KUKA KRL program: EPS_2_251825_SA29_A_20260116064109.src

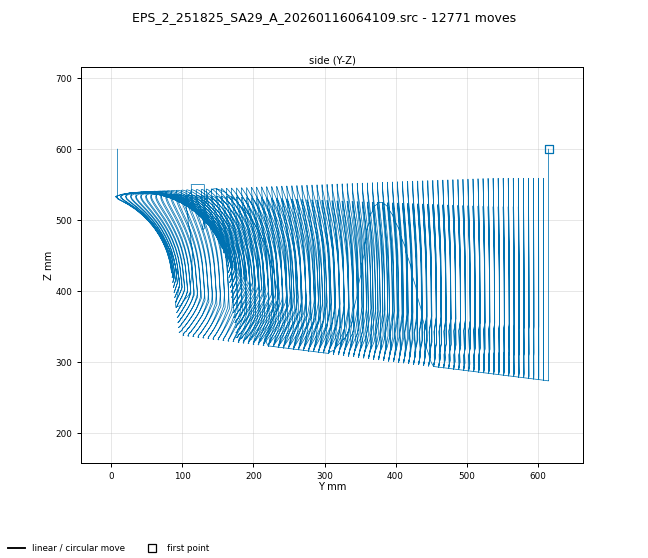
[picture p0: tool path of EPS_2_251825_SA29_A_20260116064109.src, 12771 of 12773 moves have a stored position in this frame; points joined in program order, loops and branches not executed]
&ACCESS RVP
&REL 4
&COMMENT QRS 19112012
&PARAM EDITMASK = *
DEF PART()
EXT BAS (BAS_COMMAND :IN,REAL :IN )
INT I
BAS (#INITMOV,0 )

;KUKA QRS Post kuka4.cps  Date:22-06-2017 !

File_ID=2988

QRS_PRE_INIT()

;Init var - Until changes are made in qrs_pre_init
Outlet_Square_prg=0
Inlet_1_Square_prg=0
Inlet_2_Square_prg=0
Inlet_3_Square_prg=0
Inlet_4_Square_prg=0
Inlet_5_Square_prg=0

Outlet_1={X 0.000, Y 535.490, Z 458.500, B 0.000, E1 0.000 }
Inlet_1={X 0.000, Y 538.340, Z 418.500, B 0.000, E1 195.000 }
Outlet_1_type=201
Inlet_1_type=201
;QRS#1=Sidecore dimensions
;QRS#2=200-8" PVC SDR 35
;QRS#3=200-8" PVC SDR 35
;QRS#4=
;QRS#5=
;QRS#6=
;QRS#7=
;QRS#8=
;QRS#9=12-08 PSX
;QRS#10=12-08 PSX
;QRS#11=
;QRS#12=
;QRS#13=
;QRS#14=
;QRS#15=
;QRS#16=1220x127x838 2,75'
;QRS#17=EPS Height
;QRS#18=559
;QRS#19=*
;QRS#20= UPDATED VERSION 22-06-2017
;QRS#21=*
Outlet_Square=0100
Inlet_1_Square=0100
Inlet_2_Square=0
Inlet_3_Square=0
Inlet_4_Square=0
Inlet_5_Square=0
Mill_Square=1
Outlet_Square_Prg=204
Inlet_1_Square_prg=204

QRS_INIT()

$ADVANCE=5

; T1
PTP {E1 173.613,E2 173.613}
PTP {X 0,Y 615.498,A -85,B 0,C 180,E1 173.613,E2 173.613,E3 0,E4 0,E5 0,E6 0}
QRS_SPEED_INIT()
LIN {X 0,Y 615.498,Z 600,A -85,B 0,C 180,E1 173.613,E2 173.613,E3 0,E4 0,E5 0,E6 0} C_VEL
LIN {X 0,Y 615.498,Z 283.876,A -85,B 0,C 180,E1 173.613,E2 173.613} C_VEL
LIN {X 0,Y 615.498,Z 275.694,A -85,B 0,C 180,E1 173.613,E2 173.613} C_VEL
LIN {X 0,Y 615.484,Z 273.694,A -85,B 0,C 180,E1 173.427,E2 173.427} C_VEL
LIN {X 0,Y 615.492,Z 273.68,A -85,B 0,C 180,E1 170.801,E2 170.801} C_VEL
LIN {X 0,Y 615.47,Z 273.687,A -85,B 0,C 180,E1 168.139,E2 168.139} C_VEL
LIN {X 0,Y 615.487,Z 273.702,A -85,B 0,C 180,E1 165.451,E2 165.451} C_VEL
LIN {X 0,Y 615.479,Z 273.686,A -85,B 0,C 180,E1 162.729,E2 162.729} C_VEL
LIN {X 0,Y 615.473,Z 273.685,A -85,B 0,C 180,E1 159.967,E2 159.967} C_VEL
LIN {X 0,Y 615.486,Z 273.703,A -85,B 0,C 180,E1 157.156,E2 157.156} C_VEL
LIN {X 0,Y 615.489,Z 273.681,A -85,B 0,C 180,E1 154.284,E2 154.284} C_VEL
LIN {X 0,Y 615.471,Z 273.688,A -85,B 0,C 180,E1 151.553,E2 151.553} C_VEL
LIN {X 0,Y 615.486,Z 273.702,A -85,B 0,C 180,E1 148.915,E2 148.915} C_VEL
LIN {X 0,Y 615.491,Z 273.68,A -85,B 0,C 180,E1 145.978,E2 145.978} C_VEL
LIN {X 0,Y 615.473,Z 273.692,A -85,B 0,C 180,E1 143.066,E2 143.066} C_VEL
LIN {X 0,Y 615.481,Z 273.692,A -85,B 0,C 180,E1 140.249,E2 140.249} C_VEL
LIN {X 0,Y 615.494,Z 273.679,A -85,B 0,C 180,E1 137.648,E2 137.648} C_VEL
LIN {X 0,Y 615.471,Z 273.689,A -85,B 0,C 180,E1 134.93,E2 134.93} C_VEL
LIN {X 0,Y 615.481,Z 273.695,A -85,B 0,C 180,E1 132.08,E2 132.08} C_VEL
LIN {X 0,Y 615.479,Z 273.688,A -85,B 0,C 180,E1 129.751,E2 129.751} C_VEL
LIN {X 0,Y 615.477,Z 273.684,A -85,B 0,C 180,E1 126.935,E2 126.935} C_VEL
LIN {X 0,Y 615.495,Z 273.7,A -85,B 0,C 180,E1 124.022,E2 124.022} C_VEL
LIN {X 0,Y 615.481,Z 273.682,A -85,B 0,C 180,E1 121.085,E2 121.085} C_VEL
LIN {X 0,Y 615.471,Z 273.688,A -85,B 0,C 180,E1 118.448,E2 118.448} C_VEL
LIN {X 0,Y 615.494,Z 273.699,A -85,B 0,C 180,E1 115.716,E2 115.716} C_VEL
LIN {X 0,Y 615.491,Z 273.68,A -85,B 0,C 180,E1 112.845,E2 112.845} C_VEL
LIN {X 0,Y 615.472,Z 273.691,A -85,B 0,C 180,E1 110.034,E2 110.034} C_VEL
LIN {X 0,Y 615.484,Z 273.694,A -85,B 0,C 180,E1 107.271,E2 107.271} C_VEL
LIN {X 0,Y 615.492,Z 273.68,A -85,B 0,C 180,E1 104.55,E2 104.55} C_VEL
LIN {X 0,Y 615.472,Z 273.689,A -85,B 0,C 180,E1 101.862,E2 101.862} C_VEL
LIN {X 0,Y 615.496,Z 273.699,A -85,B 0,C 180,E1 99.2,E2 99.2} C_VEL
LIN {X 0,Y 615.478,Z 273.686,A -85,B 0,C 180,E1 96.558,E2 96.558} C_VEL
LIN {X 0,Y 615.475,Z 273.685,A -85,B 0,C 180,E1 93.766,E2 93.766} C_VEL
LIN {X 0,Y 615.472,Z 273.814,A -85,B 0,C 180,E1 93.602,E2 93.602} C_VEL
LIN {X 0,Y 615.48,Z 289.251,A -85,B 0,C 180,E1 90.982,E2 90.982} C_VEL
LIN {X 0,Y 615.46,Z 304.876,A -85,B 0,C 180,E1 88.365,E2 88.365} C_VEL
LIN {X 0,Y 615.492,Z 308.179,A -85,B 0,C 180,E1 87.813,E2 87.813} C_VEL
LIN {X 0,Y 615.438,Z 414.942,A -85,B 0,C 180,E1 86.543,E2 86.543} C_VEL
LIN {X 0,Y 615.452,Z 427.227,A -85,B 0,C 180,E1 86.277,E2 86.277} C_VEL
LIN {X 0,Y 615.49,Z 439.928,A -85,B 0,C 180,E1 85.868,E2 85.868} C_VEL
LIN {X 0,Y 615.468,Z 452.119,A -85,B 0,C 180,E1 85.334,E2 85.334} C_VEL
LIN {X 0,Y 615.471,Z 463.598,A -85,B 0,C 180,E1 84.678,E2 84.678} C_VEL
LIN {X 0,Y 615.498,Z 473.921,A -85,B 0,C 180,E1 83.938,E2 83.938} C_VEL
LIN {X 0,Y 615.498,Z 481.714,A -85,B 0,C 180,E1 83.256,E2 83.256} C_VEL
LIN {X 0,Y 615.497,Z 489.534,A -85,B 0,C 180,E1 82.456,E2 82.456} C_VEL
LIN {X 0,Y 615.494,Z 497.406,A -85,B 0,C 180,E1 81.465,E2 81.465} C_VEL
LIN {X 0,Y 615.497,Z 503.699,A -85,B 0,C 180,E1 80.471,E2 80.471} C_VEL
LIN {X 0,Y 615.497,Z 508.721,A -85,B 0,C 180,E1 79.474,E2 79.474} C_VEL
LIN {X 0,Y 615.496,Z 512.609,A -85,B 0,C 180,E1 78.475,E2 78.475} C_VEL
LIN {X 0,Y 615.496,Z 515.466,A -85,B 0,C 180,E1 77.471,E2 77.471} C_VEL
LIN {X 0,Y 615.496,Z 516.804,A -85,B 0,C 180,E1 76.8,E2 76.8} C_VEL
LIN {X 0,Y 615.496,Z 517.816,A -85,B 0,C 180,E1 76.064,E2 76.064} C_VEL
LIN {X 0,Y 615.497,Z 518.274,A -85,B 0,C 180,E1 75.452,E2 75.452} C_VEL
LIN {X 0,Y 615.496,Z 518.351,A -85,B 0,C 180,E1 74.775,E2 74.775} C_VEL
LIN {X 0,Y 615.495,Z 517.486,A -85,B 0,C 180,E1 73.566,E2 73.566} C_VEL
LIN {X 0,Y 615.495,Z 516.099,A -85,B 0,C 180,E1 72.731,E2 72.731} C_VEL
LIN {X 0,Y 615.497,Z 514.451,A -85,B 0,C 180,E1 72.045,E2 72.045} C_VEL
LIN {X 0,Y 615.496,Z 511.079,A -85,B 0,C 180,E1 71.01,E2 71.01} C_VEL
LIN {X 0,Y 615.495,Z 506.514,A -85,B 0,C 180,E1 69.969,E2 69.969} C_VEL
LIN {X 0,Y 615.495,Z 500.595,A -85,B 0,C 180,E1 68.921,E2 68.921} C_VEL
LIN {X 0,Y 615.497,Z 492.996,A -85,B 0,C 180,E1 67.865,E2 67.865} C_VEL
LIN {X 0,Y 615.498,Z 485.049,A -85,B 0,C 180,E1 66.98,E2 66.98} C_VEL
LIN {X 0,Y 615.498,Z 476.915,A -85,B 0,C 180,E1 66.218,E2 66.218} C_VEL
LIN {X 0,Y 615.495,Z 467.048,A -85,B 0,C 180,E1 65.46,E2 65.46} C_VEL
LIN {X 0,Y 615.48,Z 456.212,A -85,B 0,C 180,E1 64.793,E2 64.793} C_VEL
LIN {X 0,Y 615.489,Z 443.762,A -85,B 0,C 180,E1 64.195,E2 64.195} C_VEL
LIN {X 0,Y 615.47,Z 431.051,A -85,B 0,C 180,E1 63.739,E2 63.739} C_VEL
LIN {X 0,Y 615.474,Z 418.085,A -85,B 0,C 180,E1 63.425,E2 63.425} C_VEL
LIN {X 0,Y 615.489,Z 400.248,A -85,B 0,C 180,E1 63.181,E2 63.181} C_VEL
LIN {X 0,Y 615.471,Z 308.115,A -85,B 0,C 180,E1 62.086,E2 62.086} C_VEL
LIN {X 0,Y 615.45,Z 292.43,A -85,B 0,C 180,E1 59.46,E2 59.46} C_VEL
LIN {X 0,Y 615.467,Z 276.486,A -85,B 0,C 180,E1 56.764,E2 56.764} C_VEL
LIN {X 0,Y 615.421,Z 273.7,A -85,B 0,C 180,E1 56.286,E2 56.286} C_VEL
LIN {X 0,Y 615.406,Z 273.7,A -85,B 0,C 180,E1 53.571,E2 53.571} C_VEL
LIN {X 0,Y 615.464,Z 273.7,A -85,B 0,C 180,E1 50.941,E2 50.941} C_VEL
LIN {X 0,Y 615.484,Z 273.698,A -85,B 0,C 180,E1 48.528,E2 48.528} C_VEL
LIN {X 0,Y 615.417,Z 273.698,A -85,B 0,C 180,E1 45.846,E2 45.846} C_VEL
LIN {X 0,Y 615.417,Z 273.699,A -85,B 0,C 180,E1 43.251,E2 43.251} C_VEL
LIN {X 0,Y 615.479,Z 273.7,A -85,B 0,C 180,E1 40.607,E2 40.607} C_VEL
LIN {X 0,Y 615.46,Z 273.695,A -85,B 0,C 180,E1 38.011,E2 38.011} C_VEL
LIN {X 0,Y 615.43,Z 273.695,A -85,B 0,C 180,E1 35.62,E2 35.62} C_VEL
LIN {X 0,Y 615.419,Z 273.696,A -85,B 0,C 180,E1 33.24,E2 33.24} C_VEL
LIN {X 0,Y 615.426,Z 273.697,A -85,B 0,C 180,E1 30.923,E2 30.923} C_VEL
LIN {X 0,Y 615.462,Z 273.699,A -85,B 0,C 180,E1 28.449,E2 28.449} C_VEL
LIN {X 0,Y 615.46,Z 273.692,A -85,B 0,C 180,E1 25.567,E2 25.567} C_VEL
LIN {X 0,Y 615.467,Z 273.691,A -85,B 0,C 180,E1 23.557,E2 23.557} C_VEL
LIN {X 0,Y 615.461,Z 273.691,A -85,B 0,C 180,E1 21.433,E2 21.433} C_VEL
LIN {X 0,Y 615.459,Z 273.69,A -85,B 0,C 180,E1 19.339,E2 19.339} C_VEL
LIN {X 0,Y 615.456,Z 273.691,A -85,B 0,C 180,E1 17.271,E2 17.271} C_VEL
LIN {X 0,Y 615.463,Z 273.689,A -85,B 0,C 180,E1 15.227,E2 15.227} C_VEL
LIN {X 0,Y 615.468,Z 273.688,A -85,B 0,C 180,E1 13.202,E2 13.202} C_VEL
LIN {X 0,Y 615.437,Z 273.693,A -85,B 0,C 180,E1 10.528,E2 10.528} C_VEL
LIN {X 0,Y 615.475,Z 273.698,A -85,B 0,C 180,E1 7.876,E2 7.876} C_VEL
LIN {X 0,Y 615.493,Z 273.688,A -85,B 0,C 180,E1 5.241,E2 5.241} C_VEL
LIN {X 0,Y 615.452,Z 273.689,A -85,B 0,C 180,E1 2.618,E2 2.618} C_VEL
LIN {X 0,Y 615.456,Z 273.688,A -85,B 0,C 180,E1 0.654,E2 0.654} C_VEL
LIN {X 0,Y 615.468,Z 273.686,A -85,B 0,C 180,E1 -1.309,E2 -1.309} C_VEL
LIN {X 0,Y 615.479,Z 273.685,A -85,B 0,C 180,E1 -3.273,E2 -3.273} C_VEL
LIN {X 0,Y 615.449,Z 273.691,A -85,B 0,C 180,E1 -5.899,E2 -5.899} C_VEL
LIN {X 0,Y 615.48,Z 273.698,A -85,B 0,C 180,E1 -8.537,E2 -8.537} C_VEL
LIN {X 0,Y 615.492,Z 273.687,A -85,B 0,C 180,E1 -11.193,E2 -11.193} C_VEL
LIN {X 0,Y 615.459,Z 273.687,A -85,B 0,C 180,E1 -13.929,E2 -13.929} C_VEL
LIN {X 0,Y 615.469,Z 273.696,A -85,B 0,C 180,E1 -16.587,E2 -16.587} C_VEL
LIN {X 0,Y 615.489,Z 273.689,A -85,B 0,C 180,E1 -19.338,E2 -19.338} C_VEL
LIN {X 0,Y 615.464,Z 273.686,A -85,B 0,C 180,E1 -22.138,E2 -22.138} C_VEL
LIN {X 0,Y 615.463,Z 273.687,A -85,B 0,C 180,E1 -24.273,E2 -24.273} C_VEL
LIN {X 0,Y 615.489,Z 273.699,A -85,B 0,C 180,E1 -27.049,E2 -27.049} C_VEL
LIN {X 0,Y 615.489,Z 273.684,A -85,B 0,C 180,E1 -29.798,E2 -29.798} C_VEL
LIN {X 0,Y 615.47,Z 273.685,A -85,B 0,C 180,E1 -32.459,E2 -32.459} C_VEL
LIN {X 0,Y 615.467,Z 273.691,A -85,B 0,C 180,E1 -34.817,E2 -34.817} C_VEL
LIN {X 0,Y 615.482,Z 273.698,A -85,B 0,C 180,E1 -37.243,E2 -37.243} C_VEL
LIN {X 0,Y 615.483,Z 273.685,A -85,B 0,C 180,E1 -40.091,E2 -40.091} C_VEL
LIN {X 0,Y 615.495,Z 273.68,A -85,B 0,C 180,E1 -42.353,E2 -42.353} C_VEL
LIN {X 0,Y 615.472,Z 273.69,A -85,B 0,C 180,E1 -45.07,E2 -45.07} C_VEL
LIN {X 0,Y 615.482,Z 273.694,A -85,B 0,C 180,E1 -47.921,E2 -47.921} C_VEL
LIN {X 0,Y 615.477,Z 273.688,A -85,B 0,C 180,E1 -50.251,E2 -50.251} C_VEL
LIN {X 0,Y 615.479,Z 273.684,A -85,B 0,C 180,E1 -53.065,E2 -53.065} C_VEL
LIN {X 0,Y 615.488,Z 273.697,A -85,B 0,C 180,E1 -55.98,E2 -55.98} C_VEL
LIN {X 0,Y 615.48,Z 273.682,A -85,B 0,C 180,E1 -58.916,E2 -58.916} C_VEL
LIN {X 0,Y 615.479,Z 273.69,A -85,B 0,C 180,E1 -61.552,E2 -61.552} C_VEL
LIN {X 0,Y 615.48,Z 273.695,A -85,B 0,C 180,E1 -64.285,E2 -64.285} C_VEL
LIN {X 0,Y 615.489,Z 273.68,A -85,B 0,C 180,E1 -67.157,E2 -67.157} C_VEL
LIN {X 0,Y 615.487,Z 273.758,A -85,B 0,C 180,E1 -67.438,E2 -67.438} C_VEL
LIN {X 0,Y 615.455,Z 293.701,A -85,B 0,C 180,E1 -70.141,E2 -70.141} C_VEL
LIN {X 0,Y 615.472,Z 313.086,A -85,B 0,C 180,E1 -72.73,E2 -72.73} C_VEL
LIN {X 0,Y 615.493,Z 334.924,A -85,B 0,C 180,E1 -75.607,E2 -75.607} C_VEL
LIN {X 0,Y 615.471,Z 346.477,A -85,B 0,C 180,E1 -77.114,E2 -77.114} C_VEL
LIN {X 0,Y 615.457,Z 454.9,A -85,B 0,C 180,E1 -78.411,E2 -78.411} C_VEL
LIN {X 0,Y 615.456,Z 467.391,A -85,B 0,C 180,E1 -78.682,E2 -78.682} C_VEL
LIN {X 0,Y 615.483,Z 480.688,A -85,B 0,C 180,E1 -79.116,E2 -79.116} C_VEL
LIN {X 0,Y 615.492,Z 492.498,A -85,B 0,C 180,E1 -79.641,E2 -79.641} C_VEL
LIN {X 0,Y 615.483,Z 504.013,A -85,B 0,C 180,E1 -80.305,E2 -80.305} C_VEL
LIN {X 0,Y 615.499,Z 514.355,A -85,B 0,C 180,E1 -81.051,E2 -81.051} C_VEL
LIN {X 0,Y 615.497,Z 522.703,A -85,B 0,C 180,E1 -81.795,E2 -81.795} C_VEL
LIN {X 0,Y 615.498,Z 530.615,A -85,B 0,C 180,E1 -82.621,E2 -82.621} C_VEL
LIN {X 0,Y 615.491,Z 538.211,A -85,B 0,C 180,E1 -83.609,E2 -83.609} C_VEL
LIN {X 0,Y 615.498,Z 545.21,A -85,B 0,C 180,E1 -84.76,E2 -84.76} C_VEL
LIN {X 0,Y 615.493,Z 549.856,A -85,B 0,C 180,E1 -85.745,E2 -85.745} C_VEL
LIN {X 0,Y 615.494,Z 553.402,A -85,B 0,C 180,E1 -86.728,E2 -86.728} C_VEL
LIN {X 0,Y 615.497,Z 555.235,A -85,B 0,C 180,E1 -87.383,E2 -87.383} C_VEL
LIN {X 0,Y 615.497,Z 556.61,A -85,B 0,C 180,E1 -88.038,E2 -88.038} C_VEL
LIN {X 0,Y 615.496,Z 558.174,A -85,B 0,C 180,E1 -89.347,E2 -89.347} C_VEL
LIN {X 0,Y 615.494,Z 558.389,A -85,B 0,C 180,E1 -90.001,E2 -90.001} C_VEL
LIN {X 0,Y 615.495,Z 557.579,A -85,B 0,C 180,E1 -91.31,E2 -91.31} C_VEL
LIN {X 0,Y 615.497,Z 556.607,A -85,B 0,C 180,E1 -91.964,E2 -91.964} C_VEL
LIN {X 0,Y 615.497,Z 555.23,A -85,B 0,C 180,E1 -92.619,E2 -92.619} C_VEL
LIN {X 0,Y 615.496,Z 552.346,A -85,B 0,C 180,E1 -93.602,E2 -93.602} C_VEL
LIN {X 0,Y 615.498,Z 548.438,A -85,B 0,C 180,E1 -94.585,E2 -94.585} C_VEL
LIN {X 0,Y 615.499,Z 543.4,A -85,B 0,C 180,E1 -95.571,E2 -95.571} C_VEL
LIN {X 0,Y 615.49,Z 536.913,A -85,B 0,C 180,E1 -96.578,E2 -96.578} C_VEL
LIN {X 0,Y 615.497,Z 529.125,A -85,B 0,C 180,E1 -97.546,E2 -97.546} C_VEL
LIN {X 0,Y 615.498,Z 519.247,A -85,B 0,C 180,E1 -98.537,E2 -98.537} C_VEL
LIN {X 0,Y 615.495,Z 508.853,A -85,B 0,C 180,E1 -99.365,E2 -99.365} C_VEL
LIN {X 0,Y 615.482,Z 498.561,A -85,B 0,C 180,E1 -100.029,E2 -100.029} C_VEL
LIN {X 0,Y 615.495,Z 487.122,A -85,B 0,C 180,E1 -100.617,E2 -100.617} C_VEL
LIN {X 0,Y 615.466,Z 475.341,A -85,B 0,C 180,E1 -101.078,E2 -101.078} C_VEL
LIN {X 0,Y 615.455,Z 462.209,A -85,B 0,C 180,E1 -101.445,E2 -101.445} C_VEL
LIN {X 0,Y 615.461,Z 448.878,A -85,B 0,C 180,E1 -101.674,E2 -101.674} C_VEL
LIN {X 0,Y 615.471,Z 346.462,A -85,B 0,C 180,E1 -102.888,E2 -102.888} C_VEL
LIN {X 0,Y 615.455,Z 325.984,A -85,B 0,C 180,E1 -105.567,E2 -105.567} C_VEL
LIN {X 0,Y 615.481,Z 305.471,A -85,B 0,C 180,E1 -108.282,E2 -108.282} C_VEL
LIN {X 0,Y 615.468,Z 283.338,A -85,B 0,C 180,E1 -111.258,E2 -111.258} C_VEL
LIN {X 0,Y 615.489,Z 273.682,A -85,B 0,C 180,E1 -112.594,E2 -112.594} C_VEL
LIN {X 0,Y 615.485,Z 273.681,A -85,B 0,C 180,E1 -114.993,E2 -114.993} C_VEL
LIN {X 0,Y 615.483,Z 273.698,A -85,B 0,C 180,E1 -117.916,E2 -117.916} C_VEL
LIN {X 0,Y 615.486,Z 273.682,A -85,B 0,C 180,E1 -120.921,E2 -120.921} C_VEL
LIN {X 0,Y 615.47,Z 273.686,A -85,B 0,C 180,E1 -123.531,E2 -123.531} C_VEL
LIN {X 0,Y 615.487,Z 273.7,A -85,B 0,C 180,E1 -126.425,E2 -126.425} C_VEL
LIN {X 0,Y 615.482,Z 273.685,A -85,B 0,C 180,E1 -129.061,E2 -129.061} C_VEL
LIN {X 0,Y 615.491,Z 273.68,A -85,B 0,C 180,E1 -131.474,E2 -131.474} C_VEL
LIN {X 0,Y 615.47,Z 273.691,A -85,B 0,C 180,E1 -134.152,E2 -134.152} C_VEL
LIN {X 0,Y 615.484,Z 273.693,A -85,B 0,C 180,E1 -136.954,E2 -136.954} C_VEL
LIN {X 0,Y 615.484,Z 273.684,A -85,B 0,C 180,E1 -139.393,E2 -139.393} C_VEL
LIN {X 0,Y 615.478,Z 273.683,A -85,B 0,C 180,E1 -141.99,E2 -141.99} C_VEL
LIN {X 0,Y 615.469,Z 273.689,A -85,B 0,C 180,E1 -144.383,E2 -144.383} C_VEL
LIN {X 0,Y 615.478,Z 273.695,A -85,B 0,C 180,E1 -146.763,E2 -146.763} C_VEL
LIN {X 0,Y 615.49,Z 273.702,A -85,B 0,C 180,E1 -149.08,E2 -149.08} C_VEL
LIN {X 0,Y 615.484,Z 273.681,A -85,B 0,C 180,E1 -152.085,E2 -152.085} C_VEL
LIN {X 0,Y 615.476,Z 273.683,A -85,B 0,C 180,E1 -154.434,E2 -154.434} C_VEL
LIN {X 0,Y 615.482,Z 273.696,A -85,B 0,C 180,E1 -157.155,E2 -157.155} C_VEL
LIN {X 0,Y 615.481,Z 273.687,A -85,B 0,C 180,E1 -159.967,E2 -159.967} C_VEL
LIN {X 0,Y 615.473,Z 273.684,A -85,B 0,C 180,E1 -162.729,E2 -162.729} C_VEL
LIN {X 0,Y 615.484,Z 273.697,A -85,B 0,C 180,E1 -165.451,E2 -165.451} C_VEL
LIN {X 0,Y 615.48,Z 273.69,A -85,B 0,C 180,E1 -168.139,E2 -168.139} C_VEL
LIN {X 0,Y 615.489,Z 273.68,A -85,B 0,C 180,E1 -170.801,E2 -170.801} C_VEL
LIN {X 0,Y 615.471,Z 273.691,A -85,B 0,C 180,E1 -173.443,E2 -173.443} C_VEL
LIN {X 0,Y 615.488,Z 273.699,A -85,B 0,C 180,E1 -176.071,E2 -176.071} C_VEL
LIN {X 0,Y 615.483,Z 273.684,A -85,B 0,C 180,E1 -178.691,E2 -178.691} C_VEL
LIN {X 0,Y 615.478,Z 273.683,A -85,B 0,C 180,E1 -181.308,E2 -181.308} C_VEL
LIN {X 0,Y 615.476,Z 273.694,A -85,B 0,C 180,E1 -183.928,E2 -183.928} C_VEL
LIN {X 0,Y 615.484,Z 273.694,A -85,B 0,C 180,E1 -186.573,E2 -186.573} C_VEL
LIN {X 0,Y 614.811,Z 273.83,A -85,B 0,C 180,E1 -187.118,E2 -187.118} C_VEL
LIN {X 0,Y 611.983,Z 274.251,A -85,B 0,C 180,E1 -188.004,E2 -188.004} C_VEL
LIN {X 0,Y 609.592,Z 274.558,A -85,B 0,C 180,E1 -188.717,E2 -188.717} C_VEL
LIN {X 0,Y 608.552,Z 274.675,A -85,B 0,C 180,E1 -189.267,E2 -189.267} C_VEL
LIN {X 0,Y 608.459,Z 274.685,A -85,B 0,C 180,E1 -189.453,E2 -189.453} C_VEL
LIN {X 0,Y 608.452,Z 274.689,A -85,B 0,C 180,E1 -192,E2 -192} C_VEL
LIN {X 0,Y 608.475,Z 274.693,A -85,B 0,C 180,E1 -194.72,E2 -194.72} C_VEL
LIN {X 0,Y 608.446,Z 274.688,A -85,B 0,C 180,E1 -197.477,E2 -197.477} C_VEL
LIN {X 0,Y 608.446,Z 274.687,A -85,B 0,C 180,E1 -199.571,E2 -199.571} C_VEL
LIN {X 0,Y 608.46,Z 274.685,A -85,B 0,C 180,E1 -201.692,E2 -201.692} C_VEL
LIN {X 0,Y 608.448,Z 274.692,A -85,B 0,C 180,E1 -204.571,E2 -204.571} C_VEL
LIN {X 0,Y 608.482,Z 274.69,A -85,B 0,C 180,E1 -207.207,E2 -207.207} C_VEL
LIN {X 0,Y 608.468,Z 274.684,A -85,B 0,C 180,E1 -209.971,E2 -209.971} C_VEL
LIN {X 0,Y 608.453,Z 274.692,A -85,B 0,C 180,E1 -212.88,E2 -212.88} C_VEL
LIN {X 0,Y 608.436,Z 274.7,A -85,B 0,C 180,E1 -215.278,E2 -215.278} C_VEL
LIN {X 0,Y 608.468,Z 274.689,A -85,B 0,C 180,E1 -217.746,E2 -217.746} C_VEL
LIN {X 0,Y 608.446,Z 274.687,A -85,B 0,C 180,E1 -220.328,E2 -220.328} C_VEL
LIN {X 0,Y 608.441,Z 274.69,A -85,B 0,C 180,E1 -222.961,E2 -222.961} C_VEL
LIN {X 0,Y 608.453,Z 274.695,A -85,B 0,C 180,E1 -225.736,E2 -225.736} C_VEL
LIN {X 0,Y 608.462,Z 274.685,A -85,B 0,C 180,E1 -228.658,E2 -228.658} C_VEL
LIN {X 0,Y 608.469,Z 274.695,A -85,B 0,C 180,E1 -231.759,E2 -231.759} C_VEL
LIN {X 0,Y 608.447,Z 274.697,A -85,B 0,C 180,E1 -233.954,E2 -233.954} C_VEL
LIN {X 0,Y 608.45,Z 274.691,A -85,B 0,C 180,E1 -236.328,E2 -236.328} C_VEL
LIN {X 0,Y 608.448,Z 274.688,A -85,B 0,C 180,E1 -238.732,E2 -238.732} C_VEL
LIN {X 0,Y 608.464,Z 274.686,A -85,B 0,C 180,E1 -241.382,E2 -241.382} C_VEL
LIN {X 0,Y 608.444,Z 274.694,A -85,B 0,C 180,E1 -243.964,E2 -243.964} C_VEL
LIN {X 0,Y 608.454,Z 274.688,A -85,B 0,C 180,E1 -246.875,E2 -246.875} C_VEL
LIN {X 0,Y 608.455,Z 274.687,A -85,B 0,C 180,E1 -249.725,E2 -249.725} C_VEL
LIN {X 0,Y 608.442,Z 274.689,A -85,B 0,C 180,E1 -251.827,E2 -251.827} C_VEL
LIN {X 0,Y 608.466,Z 274.696,A -85,B 0,C 180,E1 -254.593,E2 -254.593} C_VEL
LIN {X 0,Y 608.475,Z 274.685,A -85,B 0,C 180,E1 -257.322,E2 -257.322} C_VEL
LIN {X 0,Y 608.445,Z 274.688,A -85,B 0,C 180,E1 -260.022,E2 -260.022} C_VEL
LIN {X 0,Y 608.464,Z 274.694,A -85,B 0,C 180,E1 -262.7,E2 -262.7} C_VEL
LIN {X 0,Y 608.448,Z 274.691,A -85,B 0,C 180,E1 -265.361,E2 -265.361} C_VEL
LIN {X 0,Y 608.459,Z 274.691,A -85,B 0,C 180,E1 -266.315,E2 -266.315} C_VEL
LIN {X 0,Y 608.494,Z 288.467,A -85,B 0,C 180,E1 -268.675,E2 -268.675} C_VEL
LIN {X 0,Y 608.44,Z 304.132,A -85,B 0,C 180,E1 -271.323,E2 -271.323} C_VEL
LIN {X 0,Y 608.493,Z 308.629,A -85,B 0,C 180,E1 -272.047,E2 -272.047} C_VEL
LIN {X 0,Y 608.484,Z 415.486,A -85,B 0,C 180,E1 -273.33,E2 -273.33} C_VEL
LIN {X 0,Y 608.496,Z 429.112,A -85,B 0,C 180,E1 -273.641,E2 -273.641} C_VEL
LIN {X 0,Y 608.528,Z 441.372,A -85,B 0,C 180,E1 -274.055,E2 -274.055} C_VEL
LIN {X 0,Y 608.474,Z 452.439,A -85,B 0,C 180,E1 -274.553,E2 -274.553} C_VEL
LIN {X 0,Y 608.457,Z 463.926,A -85,B 0,C 180,E1 -275.218,E2 -275.218} C_VEL
LIN {X 0,Y 608.498,Z 474.271,A -85,B 0,C 180,E1 -275.965,E2 -275.965} C_VEL
LIN {X 0,Y 608.478,Z 481.861,A -85,B 0,C 180,E1 -276.631,E2 -276.631} C_VEL
LIN {X 0,Y 608.47,Z 489.951,A -85,B 0,C 180,E1 -277.465,E2 -277.465} C_VEL
LIN {X 0,Y 608.44,Z 497.87,A -85,B 0,C 180,E1 -278.468,E2 -278.468} C_VEL
LIN {X 0,Y 608.437,Z 503.247,A -85,B 0,C 180,E1 -279.305,E2 -279.305} C_VEL
LIN {X 0,Y 608.459,Z 508.516,A -85,B 0,C 180,E1 -280.312,E2 -280.312} C_VEL
LIN {X 0,Y 608.427,Z 512.617,A -85,B 0,C 180,E1 -281.324,E2 -281.324} C_VEL
LIN {X 0,Y 608.439,Z 514.749,A -85,B 0,C 180,E1 -281.999,E2 -281.999} C_VEL
LIN {X 0,Y 608.419,Z 516.43,A -85,B 0,C 180,E1 -282.677,E2 -282.677} C_VEL
LIN {X 0,Y 608.438,Z 517.694,A -85,B 0,C 180,E1 -283.356,E2 -283.356} C_VEL
LIN {X 0,Y 608.421,Z 518.539,A -85,B 0,C 180,E1 -284.037,E2 -284.037} C_VEL
LIN {X 0,Y 608.418,Z 518.93,A -85,B 0,C 180,E1 -284.721,E2 -284.721} C_VEL
LIN {X 0,Y 608.418,Z 518.921,A -85,B 0,C 180,E1 -285.406,E2 -285.406} C_VEL
LIN {X 0,Y 608.423,Z 518.012,A -85,B 0,C 180,E1 -286.515,E2 -286.515} C_VEL
LIN {X 0,Y 608.42,Z 516.293,A -85,B 0,C 180,E1 -287.476,E2 -287.476} C_VEL
LIN {X 0,Y 608.428,Z 512.84,A -85,B 0,C 180,E1 -288.704,E2 -288.704} C_VEL
LIN {X 0,Y 608.434,Z 507.819,A -85,B 0,C 180,E1 -289.921,E2 -289.921} C_VEL
LIN {X 0,Y 608.45,Z 502.058,A -85,B 0,C 180,E1 -290.98,E2 -290.98} C_VEL
LIN {X 0,Y 608.454,Z 494.729,A -85,B 0,C 180,E1 -292.047,E2 -292.047} C_VEL
LIN {X 0,Y 608.456,Z 487.093,A -85,B 0,C 180,E1 -292.942,E2 -292.942} C_VEL
LIN {X 0,Y 608.481,Z 477.658,A -85,B 0,C 180,E1 -293.843,E2 -293.843} C_VEL
LIN {X 0,Y 608.493,Z 467.137,A -85,B 0,C 180,E1 -294.659,E2 -294.659} C_VEL
LIN {X 0,Y 608.48,Z 455.524,A -85,B 0,C 180,E1 -295.371,E2 -295.371} C_VEL
LIN {X 0,Y 608.517,Z 443.797,A -85,B 0,C 180,E1 -295.934,E2 -295.934} C_VEL
LIN {X 0,Y 608.515,Z 432.326,A -85,B 0,C 180,E1 -296.353,E2 -296.353} C_VEL
LIN {X 0,Y 608.539,Z 419.33,A -85,B 0,C 180,E1 -296.687,E2 -296.687} C_VEL
LIN {X 0,Y 608.539,Z 403.321,A -85,B 0,C 180,E1 -296.921,E2 -296.921} C_VEL
LIN {X 0,Y 608.431,Z 308.378,A -85,B 0,C 180,E1 -298.055,E2 -298.055} C_VEL
LIN {X 0,Y 608.451,Z 293.599,A -85,B 0,C 180,E1 -300.544,E2 -300.544} C_VEL
LIN {X 0,Y 608.454,Z 276.455,A -85,B 0,C 180,E1 -303.471,E2 -303.471} C_VEL
LIN {X 0,Y 608.403,Z 274.695,A -85,B 0,C 180,E1 -303.79,E2 -303.79} C_VEL
LIN {X 0,Y 608.375,Z 274.696,A -85,B 0,C 180,E1 -306.095,E2 -306.095} C_VEL
LIN {X 0,Y 608.375,Z 274.696,A -85,B 0,C 180,E1 -308.229,E2 -308.229} C_VEL
LIN {X 0,Y 608.39,Z 274.694,A -85,B 0,C 180,E1 -310.322,E2 -310.322} C_VEL
LIN {X 0,Y 608.379,Z 274.696,A -85,B 0,C 180,E1 -312.326,E2 -312.326} C_VEL
LIN {X 0,Y 608.394,Z 274.694,A -85,B 0,C 180,E1 -314.258,E2 -314.258} C_VEL
LIN {X 0,Y 608.412,Z 274.692,A -85,B 0,C 180,E1 -316.695,E2 -316.695} C_VEL
LIN {X 0,Y 608.391,Z 274.695,A -85,B 0,C 180,E1 -318.818,E2 -318.818} C_VEL
LIN {X 0,Y 608.405,Z 274.701,A -85,B 0,C 180,E1 -321.407,E2 -321.407} C_VEL
LIN {X 0,Y 608.428,Z 274.695,A -85,B 0,C 180,E1 -323.954,E2 -323.954} C_VEL
LIN {X 0,Y 608.428,Z 274.691,A -85,B 0,C 180,E1 -326.327,E2 -326.327} C_VEL
LIN {X 0,Y 608.415,Z 274.691,A -85,B 0,C 180,E1 -328.734,E2 -328.734} C_VEL
LIN {X 0,Y 608.441,Z 274.692,A -85,B 0,C 180,E1 -331.382,E2 -331.382} C_VEL
LIN {X 0,Y 608.456,Z 274.69,A -85,B 0,C 180,E1 -334.278,E2 -334.278} C_VEL
LIN {X 0,Y 608.412,Z 274.692,A -85,B 0,C 180,E1 -336.875,E2 -336.875} C_VEL
LIN {X 0,Y 608.425,Z 274.691,A -85,B 0,C 180,E1 -339.327,E2 -339.327} C_VEL
LIN {X 0,Y 608.436,Z 274.696,A -85,B 0,C 180,E1 -341.828,E2 -341.828} C_VEL
LIN {X 0,Y 608.454,Z 274.69,A -85,B 0,C 180,E1 -344.594,E2 -344.594} C_VEL
LIN {X 0,Y 608.435,Z 274.689,A -85,B 0,C 180,E1 -347.322,E2 -347.322} C_VEL
LIN {X 0,Y 608.444,Z 274.694,A -85,B 0,C 180,E1 -350.023,E2 -350.023} C_VEL
LIN {X 0,Y 608.475,Z 274.688,A -85,B 0,C 180,E1 -352.701,E2 -352.701} C_VEL
LIN {X 0,Y 608.418,Z 274.691,A -85,B 0,C 180,E1 -355.362,E2 -355.362} C_VEL
LIN {X 0,Y 608.446,Z 274.687,A -85,B 0,C 180,E1 -357.352,E2 -357.352} C_VEL
LIN {X 0,Y 608.443,Z 274.691,A -85,B 0,C 180,E1 -360,E2 -360} C_VEL
LIN {X 0,Y 608.485,Z 274.692,A -85,B 0,C 180,E1 -362.648,E2 -362.648} C_VEL
LIN {X 0,Y 608.461,Z 274.687,A -85,B 0,C 180,E1 -365.302,E2 -365.302} C_VEL
LIN {X 0,Y 608.449,Z 274.688,A -85,B 0,C 180,E1 -367.967,E2 -367.967} C_VEL
LIN {X 0,Y 608.458,Z 274.695,A -85,B 0,C 180,E1 -370.65,E2 -370.65} C_VEL
LIN {X 0,Y 608.461,Z 274.688,A -85,B 0,C 180,E1 -373.357,E2 -373.357} C_VEL
LIN {X 0,Y 608.438,Z 274.689,A -85,B 0,C 180,E1 -376.095,E2 -376.095} C_VEL
LIN {X 0,Y 608.445,Z 274.698,A -85,B 0,C 180,E1 -378.87,E2 -378.87} C_VEL
LIN {X 0,Y 608.459,Z 274.687,A -85,B 0,C 180,E1 -381.692,E2 -381.692} C_VEL
LIN {X 0,Y 608.441,Z 274.691,A -85,B 0,C 180,E1 -384.572,E2 -384.572} C_VEL
LIN {X 0,Y 608.478,Z 274.694,A -85,B 0,C 180,E1 -387.211,E2 -387.211} C_VEL
LIN {X 0,Y 608.467,Z 274.685,A -85,B 0,C 180,E1 -389.975,E2 -389.975} C_VEL
LIN {X 0,Y 608.446,Z 274.688,A -85,B 0,C 180,E1 -392.523,E2 -392.523} C_VEL
LIN {X 0,Y 608.461,Z 274.689,A -85,B 0,C 180,E1 -394.91,E2 -394.91} C_VEL
LIN {X 0,Y 608.467,Z 274.69,A -85,B 0,C 180,E1 -397.747,E2 -397.747} C_VEL
LIN {X 0,Y 608.447,Z 274.687,A -85,B 0,C 180,E1 -400.331,E2 -400.331} C_VEL
LIN {X 0,Y 608.441,Z 274.69,A -85,B 0,C 180,E1 -402.961,E2 -402.961} C_VEL
LIN {X 0,Y 608.451,Z 274.695,A -85,B 0,C 180,E1 -405.737,E2 -405.737} C_VEL
LIN {X 0,Y 608.462,Z 274.685,A -85,B 0,C 180,E1 -408.658,E2 -408.658} C_VEL
LIN {X 0,Y 608.461,Z 274.691,A -85,B 0,C 180,E1 -411.413,E2 -411.413} C_VEL
LIN {X 0,Y 608.471,Z 274.693,A -85,B 0,C 180,E1 -413.952,E2 -413.952} C_VEL
LIN {X 0,Y 608.457,Z 274.689,A -85,B 0,C 180,E1 -416.331,E2 -416.331} C_VEL
LIN {X 0,Y 608.456,Z 274.686,A -85,B 0,C 180,E1 -418.731,E2 -418.731} C_VEL
LIN {X 0,Y 608.468,Z 274.687,A -85,B 0,C 180,E1 -421.381,E2 -421.381} C_VEL
LIN {X 0,Y 608.439,Z 274.699,A -85,B 0,C 180,E1 -423.966,E2 -423.966} C_VEL
LIN {X 0,Y 608.463,Z 274.696,A -85,B 0,C 180,E1 -426.156,E2 -426.156} C_VEL
LIN {X 0,Y 608.505,Z 274.83,A -85,B 0,C 180,E1 -427.313,E2 -427.313} C_VEL
LIN {X 0,Y 608.524,Z 292.417,A -85,B 0,C 180,E1 -429.729,E2 -429.729} C_VEL
LIN {X 0,Y 608.51,Z 311.833,A -85,B 0,C 180,E1 -432.353,E2 -432.353} C_VEL
LIN {X 0,Y 608.496,Z 332.545,A -85,B 0,C 180,E1 -435.11,E2 -435.11} C_VEL
LIN {X 0,Y 608.465,Z 346.703,A -85,B 0,C 180,E1 -436.974,E2 -436.974} C_VEL
LIN {X 0,Y 608.521,Z 455.009,A -85,B 0,C 180,E1 -438.277,E2 -438.277} C_VEL
LIN {X 0,Y 608.491,Z 468.258,A -85,B 0,C 180,E1 -438.572,E2 -438.572} C_VEL
LIN {X 0,Y 608.51,Z 480.667,A -85,B 0,C 180,E1 -438.984,E2 -438.984} C_VEL
LIN {X 0,Y 608.514,Z 492.656,A -85,B 0,C 180,E1 -439.52,E2 -439.52} C_VEL
LIN {X 0,Y 608.471,Z 504.214,A -85,B 0,C 180,E1 -440.192,E2 -440.192} C_VEL
LIN {X 0,Y 608.485,Z 514.608,A -85,B 0,C 180,E1 -440.947,E2 -440.947} C_VEL
LIN {X 0,Y 608.459,Z 523.013,A -85,B 0,C 180,E1 -441.7,E2 -441.7} C_VEL
LIN {X 0,Y 608.47,Z 530.97,A -85,B 0,C 180,E1 -442.535,E2 -442.535} C_VEL
LIN {X 0,Y 608.436,Z 538.303,A -85,B 0,C 180,E1 -443.487,E2 -443.487} C_VEL
LIN {X 0,Y 608.45,Z 543.872,A -85,B 0,C 180,E1 -444.367,E2 -444.367} C_VEL
LIN {X 0,Y 608.432,Z 548.955,A -85,B 0,C 180,E1 -445.363,E2 -445.363} C_VEL
LIN {X 0,Y 608.449,Z 552.9,A -85,B 0,C 180,E1 -446.359,E2 -446.359} C_VEL
LIN {X 0,Y 608.425,Z 555.812,A -85,B 0,C 180,E1 -447.353,E2 -447.353} C_VEL
LIN {X 0,Y 608.442,Z 557.203,A -85,B 0,C 180,E1 -448.015,E2 -448.015} C_VEL
LIN {X 0,Y 608.438,Z 558.784,A -85,B 0,C 180,E1 -449.339,E2 -449.339} C_VEL
LIN {X 0,Y 608.434,Z 559,A -85,B 0,C 180,E1 -450.001,E2 -450.001} C_VEL
LIN {X 0,Y 608.448,Z 558.183,A -85,B 0,C 180,E1 -451.325,E2 -451.325} C_VEL
LIN {X 0,Y 608.442,Z 557.2,A -85,B 0,C 180,E1 -451.987,E2 -451.987} C_VEL
LIN {X 0,Y 608.425,Z 555.807,A -85,B 0,C 180,E1 -452.649,E2 -452.649} C_VEL
LIN {X 0,Y 608.449,Z 552.893,A -85,B 0,C 180,E1 -453.643,E2 -453.643} C_VEL
LIN {X 0,Y 608.432,Z 548.946,A -85,B 0,C 180,E1 -454.639,E2 -454.639} C_VEL
LIN {X 0,Y 608.437,Z 542.871,A -85,B 0,C 180,E1 -455.802,E2 -455.802} C_VEL
LIN {X 0,Y 608.462,Z 536.228,A -85,B 0,C 180,E1 -456.8,E2 -456.8} C_VEL
LIN {X 0,Y 608.456,Z 527.981,A -85,B 0,C 180,E1 -457.801,E2 -457.801} C_VEL
LIN {X 0,Y 608.477,Z 517.588,A -85,B 0,C 180,E1 -458.804,E2 -458.804} C_VEL
LIN {X 0,Y 608.488,Z 506.734,A -85,B 0,C 180,E1 -459.642,E2 -459.642} C_VEL
LIN {X 0,Y 608.492,Z 495.757,A -85,B 0,C 180,E1 -460.314,E2 -460.314} C_VEL
LIN {X 0,Y 608.534,Z 483.808,A -85,B 0,C 180,E1 -460.888,E2 -460.888} C_VEL
LIN {X 0,Y 608.506,Z 471.852,A -85,B 0,C 180,E1 -461.324,E2 -461.324} C_VEL
LIN {X 0,Y 608.508,Z 459.466,A -85,B 0,C 180,E1 -461.641,E2 -461.641} C_VEL
LIN {X 0,Y 608.532,Z 443.659,A -85,B 0,C 180,E1 -461.872,E2 -461.872} C_VEL
LIN {X 0,Y 608.508,Z 347.07,A -85,B 0,C 180,E1 -463.016,E2 -463.016} C_VEL
LIN {X 0,Y 608.469,Z 345.474,A -85,B 0,C 180,E1 -463.187,E2 -463.187} C_VEL
LIN {X 0,Y 608.468,Z 326.057,A -85,B 0,C 180,E1 -465.75,E2 -465.75} C_VEL
LIN {X 0,Y 608.536,Z 305.499,A -85,B 0,C 180,E1 -468.498,E2 -468.498} C_VEL
LIN {X 0,Y 608.559,Z 283.34,A -85,B 0,C 180,E1 -471.511,E2 -471.511} C_VEL
LIN {X 0,Y 608.462,Z 274.687,A -85,B 0,C 180,E1 -472.715,E2 -472.715} C_VEL
LIN {X 0,Y 608.441,Z 274.689,A -85,B 0,C 180,E1 -475.302,E2 -475.302} C_VEL
LIN {X 0,Y 608.446,Z 274.69,A -85,B 0,C 180,E1 -477.519,E2 -477.519} C_VEL
LIN {X 0,Y 608.463,Z 274.694,A -85,B 0,C 180,E1 -479.97,E2 -479.97} C_VEL
LIN {X 0,Y 608.455,Z 274.687,A -85,B 0,C 180,E1 -482.88,E2 -482.88} C_VEL
LIN {X 0,Y 608.434,Z 274.689,A -85,B 0,C 180,E1 -485.279,E2 -485.279} C_VEL
LIN {X 0,Y 608.462,Z 274.687,A -85,B 0,C 180,E1 -487.747,E2 -487.747} C_VEL
LIN {X 0,Y 608.444,Z 274.696,A -85,B 0,C 180,E1 -490.328,E2 -490.328} C_VEL
LIN {X 0,Y 608.474,Z 274.684,A -85,B 0,C 180,E1 -493.309,E2 -493.309} C_VEL
LIN {X 0,Y 608.459,Z 274.688,A -85,B 0,C 180,E1 -496.129,E2 -496.129} C_VEL
LIN {X 0,Y 608.453,Z 274.697,A -85,B 0,C 180,E1 -498.823,E2 -498.823} C_VEL
LIN {X 0,Y 608.465,Z 274.685,A -85,B 0,C 180,E1 -501.761,E2 -501.761} C_VEL
LIN {X 0,Y 608.447,Z 274.687,A -85,B 0,C 180,E1 -503.955,E2 -503.955} C_VEL
LIN {X 0,Y 608.447,Z 274.688,A -85,B 0,C 180,E1 -506.328,E2 -506.328} C_VEL
LIN {X 0,Y 608.448,Z 274.692,A -85,B 0,C 180,E1 -508.733,E2 -508.733} C_VEL
LIN {X 0,Y 608.472,Z 274.691,A -85,B 0,C 180,E1 -511.381,E2 -511.381} C_VEL
LIN {X 0,Y 608.469,Z 274.684,A -85,B 0,C 180,E1 -514.28,E2 -514.28} C_VEL
LIN {X 0,Y 608.447,Z 274.69,A -85,B 0,C 180,E1 -516.876,E2 -516.876} C_VEL
LIN {X 0,Y 608.461,Z 274.691,A -85,B 0,C 180,E1 -519.726,E2 -519.726} C_VEL
LIN {X 0,Y 608.447,Z 274.692,A -85,B 0,C 180,E1 -521.828,E2 -521.828} C_VEL
LIN {X 0,Y 608.464,Z 274.685,A -85,B 0,C 180,E1 -524.594,E2 -524.594} C_VEL
LIN {X 0,Y 608.47,Z 274.689,A -85,B 0,C 180,E1 -527.323,E2 -527.323} C_VEL
LIN {X 0,Y 608.451,Z 274.693,A -85,B 0,C 180,E1 -530.022,E2 -530.022} C_VEL
LIN {X 0,Y 608.465,Z 274.685,A -85,B 0,C 180,E1 -532.7,E2 -532.7} C_VEL
LIN {X 0,Y 608.44,Z 274.69,A -85,B 0,C 180,E1 -535.362,E2 -535.362} C_VEL
LIN {X 0,Y 608.468,Z 274.696,A -85,B 0,C 180,E1 -538.014,E2 -538.014} C_VEL
LIN {X 0,Y 608.474,Z 274.686,A -85,B 0,C 180,E1 -540.662,E2 -540.662} C_VEL
LIN {X 0,Y 608.478,Z 274.683,A -85,B 0,C 180,E1 -543.311,E2 -543.311} C_VEL
LIN {X 0,Y 608.448,Z 274.692,A -85,B 0,C 180,E1 -545.967,E2 -545.967} C_VEL
LIN {X 0,Y 608.457,Z 274.693,A -85,B 0,C 180,E1 -548.636,E2 -548.636} C_VEL
LIN {X 0,Y 608.459,Z 274.685,A -85,B 0,C 180,E1 -549.453,E2 -549.453} C_VEL
LIN {X 0,Y 607.771,Z 274.777,A -85,B 0,C 180,E1 -550.005,E2 -550.005} C_VEL
LIN {X 0,Y 604.913,Z 275.131,A -85,B 0,C 180,E1 -550.902,E2 -550.902} C_VEL
LIN {X 0,Y 602.514,Z 275.431,A -85,B 0,C 180,E1 -551.624,E2 -551.624} C_VEL
LIN {X 0,Y 601.488,Z 275.559,A -85,B 0,C 180,E1 -552.181,E2 -552.181} C_VEL
LIN {X 0,Y 601.406,Z 275.568,A -85,B 0,C 180,E1 -552.369,E2 -552.369} C_VEL
LIN {X 0,Y 601.43,Z 275.567,A -85,B 0,C 180,E1 -554.897,E2 -554.897} C_VEL
LIN {X 0,Y 601.433,Z 275.566,A -85,B 0,C 180,E1 -556.986,E2 -556.986} C_VEL
LIN {X 0,Y 601.4,Z 275.565,A -85,B 0,C 180,E1 -559.809,E2 -559.809} C_VEL
LIN {X 0,Y 601.42,Z 275.569,A -85,B 0,C 180,E1 -562.605,E2 -562.605} C_VEL
LIN {X 0,Y 601.401,Z 275.576,A -85,B 0,C 180,E1 -564.879,E2 -564.879} C_VEL
LIN {X 0,Y 601.419,Z 275.567,A -85,B 0,C 180,E1 -567.362,E2 -567.362} C_VEL
LIN {X 0,Y 601.432,Z 275.561,A -85,B 0,C 180,E1 -570.164,E2 -570.164} C_VEL
LIN {X 0,Y 601.416,Z 275.566,A -85,B 0,C 180,E1 -572.714,E2 -572.714} C_VEL
LIN {X 0,Y 601.389,Z 275.575,A -85,B 0,C 180,E1 -575.11,E2 -575.11} C_VEL
LIN {X 0,Y 601.437,Z 275.57,A -85,B 0,C 180,E1 -577.419,E2 -577.419} C_VEL
LIN {X 0,Y 601.403,Z 275.566,A -85,B 0,C 180,E1 -579.996,E2 -579.996} C_VEL
LIN {X 0,Y 601.412,Z 275.564,A -85,B 0,C 180,E1 -582.67,E2 -582.67} C_VEL
LIN {X 0,Y 601.402,Z 275.574,A -85,B 0,C 180,E1 -585.479,E2 -585.479} C_VEL
LIN {X 0,Y 601.425,Z 275.563,A -85,B 0,C 180,E1 -588.407,E2 -588.407} C_VEL
LIN {X 0,Y 601.403,Z 275.565,A -85,B 0,C 180,E1 -590.872,E2 -590.872} C_VEL
LIN {X 0,Y 601.4,Z 275.569,A -85,B 0,C 180,E1 -593.416,E2 -593.416} C_VEL
LIN {X 0,Y 601.434,Z 275.57,A -85,B 0,C 180,E1 -596.064,E2 -596.064} C_VEL
LIN {X 0,Y 601.421,Z 275.565,A -85,B 0,C 180,E1 -598.545,E2 -598.545} C_VEL
LIN {X 0,Y 601.424,Z 275.562,A -85,B 0,C 180,E1 -601.372,E2 -601.372} C_VEL
LIN {X 0,Y 601.401,Z 275.567,A -85,B 0,C 180,E1 -603.635,E2 -603.635} C_VEL
LIN {X 0,Y 601.42,Z 275.568,A -85,B 0,C 180,E1 -606.589,E2 -606.589} C_VEL
LIN {X 0,Y 601.428,Z 275.561,A -85,B 0,C 180,E1 -609.477,E2 -609.477} C_VEL
LIN {X 0,Y 601.392,Z 275.574,A -85,B 0,C 180,E1 -612.311,E2 -612.311} C_VEL
LIN {X 0,Y 601.408,Z 275.573,A -85,B 0,C 180,E1 -614.408,E2 -614.408} C_VEL
LIN {X 0,Y 601.42,Z 275.565,A -85,B 0,C 180,E1 -617.171,E2 -617.171} C_VEL
LIN {X 0,Y 601.425,Z 275.562,A -85,B 0,C 180,E1 -619.904,E2 -619.904} C_VEL
LIN {X 0,Y 601.441,Z 275.568,A -85,B 0,C 180,E1 -622.614,E2 -622.614} C_VEL
LIN {X 0,Y 601.417,Z 275.568,A -85,B 0,C 180,E1 -625.307,E2 -625.307} C_VEL
LIN {X 0,Y 601.448,Z 275.743,A -85,B 0,C 180,E1 -626.272,E2 -626.272} C_VEL
LIN {X 0,Y 601.474,Z 289.518,A -85,B 0,C 180,E1 -628.66,E2 -628.66} C_VEL
LIN {X 0,Y 601.396,Z 305.187,A -85,B 0,C 180,E1 -631.338,E2 -631.338} C_VEL
LIN {X 0,Y 601.405,Z 308.391,A -85,B 0,C 180,E1 -631.882,E2 -631.882} C_VEL
LIN {X 0,Y 601.663,Z 314.36,A -85,B 0,C 180,E1 -631.965,E2 -631.965} C_VEL
LIN {X 0,Y 601.543,Z 414.79,A -85,B 0,C 180,E1 -633.18,E2 -633.18} C_VEL
LIN {X 0,Y 601.552,Z 427.9,A -85,B 0,C 180,E1 -633.474,E2 -633.474} C_VEL
LIN {X 0,Y 601.555,Z 440.489,A -85,B 0,C 180,E1 -633.893,E2 -633.893} C_VEL
LIN {X 0,Y 601.496,Z 452.594,A -85,B 0,C 180,E1 -634.439,E2 -634.439} C_VEL
LIN {X 0,Y 601.441,Z 464.059,A -85,B 0,C 180,E1 -635.111,E2 -635.111} C_VEL
LIN {X 0,Y 601.465,Z 474.382,A -85,B 0,C 180,E1 -635.867,E2 -635.867} C_VEL
LIN {X 0,Y 601.409,Z 483.661,A -85,B 0,C 180,E1 -636.71,E2 -636.71} C_VEL
LIN {X 0,Y 601.416,Z 491.475,A -85,B 0,C 180,E1 -637.553,E2 -637.553} C_VEL
LIN {X 0,Y 601.385,Z 499.054,A -85,B 0,C 180,E1 -638.568,E2 -638.568} C_VEL
LIN {X 0,Y 601.343,Z 506.086,A -85,B 0,C 180,E1 -639.756,E2 -639.756} C_VEL
LIN {X 0,Y 601.353,Z 511.501,A -85,B 0,C 180,E1 -640.976,E2 -640.976} C_VEL
LIN {X 0,Y 601.341,Z 515.224,A -85,B 0,C 180,E1 -642.143,E2 -642.143} C_VEL
LIN {X 0,Y 601.325,Z 516.815,A -85,B 0,C 180,E1 -642.829,E2 -642.829} C_VEL
LIN {X 0,Y 601.346,Z 518.566,A -85,B 0,C 180,E1 -644.063,E2 -644.063} C_VEL
LIN {X 0,Y 601.314,Z 518.972,A -85,B 0,C 180,E1 -644.899,E2 -644.899} C_VEL
LIN {X 0,Y 601.324,Z 518.867,A -85,B 0,C 180,E1 -645.592,E2 -645.592} C_VEL
LIN {X 0,Y 601.323,Z 517.945,A -85,B 0,C 180,E1 -646.589,E2 -646.589} C_VEL
LIN {X 0,Y 601.318,Z 515.894,A -85,B 0,C 180,E1 -647.689,E2 -647.689} C_VEL
LIN {X 0,Y 601.343,Z 512.662,A -85,B 0,C 180,E1 -648.798,E2 -648.798} C_VEL
LIN {X 0,Y 601.335,Z 508.627,A -85,B 0,C 180,E1 -649.811,E2 -649.811} C_VEL
LIN {X 0,Y 601.379,Z 502.681,A -85,B 0,C 180,E1 -650.947,E2 -650.947} C_VEL
LIN {X 0,Y 601.375,Z 495.983,A -85,B 0,C 180,E1 -651.959,E2 -651.959} C_VEL
LIN {X 0,Y 601.402,Z 488.638,A -85,B 0,C 180,E1 -652.864,E2 -652.864} C_VEL
LIN {X 0,Y 601.43,Z 478.593,A -85,B 0,C 180,E1 -653.865,E2 -653.865} C_VEL
LIN {X 0,Y 601.47,Z 467.981,A -85,B 0,C 180,E1 -654.711,E2 -654.711} C_VEL
LIN {X 0,Y 601.47,Z 456.709,A -85,B 0,C 180,E1 -655.429,E2 -655.429} C_VEL
LIN {X 0,Y 601.528,Z 444.94,A -85,B 0,C 180,E1 -656.013,E2 -656.013} C_VEL
LIN {X 0,Y 601.545,Z 432.039,A -85,B 0,C 180,E1 -656.496,E2 -656.496} C_VEL
LIN {X 0,Y 601.586,Z 419.462,A -85,B 0,C 180,E1 -656.821,E2 -656.821} C_VEL
LIN {X 0,Y 601.616,Z 403.767,A -85,B 0,C 180,E1 -657.055,E2 -657.055} C_VEL
LIN {X 0,Y 601.566,Z 309.567,A -85,B 0,C 180,E1 -658.184,E2 -658.184} C_VEL
LIN {X 0,Y 601.403,Z 308.304,A -85,B 0,C 180,E1 -658.222,E2 -658.222} C_VEL
LIN {X 0,Y 601.461,Z 292.382,A -85,B 0,C 180,E1 -660.938,E2 -660.938} C_VEL
LIN {X 0,Y 601.435,Z 276.034,A -85,B 0,C 180,E1 -663.767,E2 -663.767} C_VEL
LIN {X 0,Y 601.356,Z 275.573,A -85,B 0,C 180,E1 -663.925,E2 -663.925} C_VEL
LIN {X 0,Y 601.36,Z 275.572,A -85,B 0,C 180,E1 -666.584,E2 -666.584} C_VEL
LIN {X 0,Y 601.378,Z 275.577,A -85,B 0,C 180,E1 -669.127,E2 -669.127} C_VEL
LIN {X 0,Y 601.388,Z 275.571,A -85,B 0,C 180,E1 -671.766,E2 -671.766} C_VEL
LIN {X 0,Y 601.352,Z 275.571,A -85,B 0,C 180,E1 -674.528,E2 -674.528} C_VEL
LIN {X 0,Y 601.406,Z 275.575,A -85,B 0,C 180,E1 -677.408,E2 -677.408} C_VEL
LIN {X 0,Y 601.372,Z 275.569,A -85,B 0,C 180,E1 -680.47,E2 -680.47} C_VEL
LIN {X 0,Y 601.37,Z 275.569,A -85,B 0,C 180,E1 -682.624,E2 -682.624} C_VEL
LIN {X 0,Y 601.365,Z 275.571,A -85,B 0,C 180,E1 -685.065,E2 -685.065} C_VEL
LIN {X 0,Y 601.413,Z 275.571,A -85,B 0,C 180,E1 -687.483,E2 -687.483} C_VEL
LIN {X 0,Y 601.415,Z 275.573,A -85,B 0,C 180,E1 -689.851,E2 -689.851} C_VEL
LIN {X 0,Y 601.367,Z 275.57,A -85,B 0,C 180,E1 -692.643,E2 -692.643} C_VEL
LIN {X 0,Y 601.368,Z 275.569,A -85,B 0,C 180,E1 -695.12,E2 -695.12} C_VEL
LIN {X 0,Y 601.399,Z 275.567,A -85,B 0,C 180,E1 -697.394,E2 -697.394} C_VEL
LIN {X 0,Y 601.386,Z 275.575,A -85,B 0,C 180,E1 -700.19,E2 -700.19} C_VEL
LIN {X 0,Y 601.389,Z 275.566,A -85,B 0,C 180,E1 -703.013,E2 -703.013} C_VEL
LIN {X 0,Y 601.402,Z 275.572,A -85,B 0,C 180,E1 -705.909,E2 -705.909} C_VEL
LIN {X 0,Y 601.422,Z 275.568,A -85,B 0,C 180,E1 -708.542,E2 -708.542} C_VEL
LIN {X 0,Y 601.386,Z 275.567,A -85,B 0,C 180,E1 -711.262,E2 -711.262} C_VEL
LIN {X 0,Y 601.375,Z 275.568,A -85,B 0,C 180,E1 -713.377,E2 -713.377} C_VEL
LIN {X 0,Y 601.391,Z 275.566,A -85,B 0,C 180,E1 -715.308,E2 -715.308} C_VEL
LIN {X 0,Y 601.415,Z 275.563,A -85,B 0,C 180,E1 -717.321,E2 -717.321} C_VEL
LIN {X 0,Y 601.413,Z 275.566,A -85,B 0,C 180,E1 -720,E2 -720} C_VEL
LIN {X 0,Y 601.448,Z 275.568,A -85,B 0,C 180,E1 -722.679,E2 -722.679} C_VEL
LIN {X 0,Y 601.421,Z 275.563,A -85,B 0,C 180,E1 -725.364,E2 -725.364} C_VEL
LIN {X 0,Y 601.417,Z 275.564,A -85,B 0,C 180,E1 -728.061,E2 -728.061} C_VEL
LIN {X 0,Y 601.421,Z 275.569,A -85,B 0,C 180,E1 -731.018,E2 -731.018} C_VEL
LIN {X 0,Y 601.407,Z 275.565,A -85,B 0,C 180,E1 -733.516,E2 -733.516} C_VEL
LIN {X 0,Y 601.417,Z 275.565,A -85,B 0,C 180,E1 -736.288,E2 -736.288} C_VEL
LIN {X 0,Y 601.408,Z 275.573,A -85,B 0,C 180,E1 -739.099,E2 -739.099} C_VEL
LIN {X 0,Y 601.397,Z 275.565,A -85,B 0,C 180,E1 -741.96,E2 -741.96} C_VEL
LIN {X 0,Y 601.423,Z 275.562,A -85,B 0,C 180,E1 -744.294,E2 -744.294} C_VEL
LIN {X 0,Y 601.448,Z 275.57,A -85,B 0,C 180,E1 -747.111,E2 -747.111} C_VEL
LIN {X 0,Y 601.438,Z 275.56,A -85,B 0,C 180,E1 -750.164,E2 -750.164} C_VEL
LIN {X 0,Y 601.41,Z 275.566,A -85,B 0,C 180,E1 -752.717,E2 -752.717} C_VEL
LIN {X 0,Y 601.399,Z 275.573,A -85,B 0,C 180,E1 -755.115,E2 -755.115} C_VEL
LIN {X 0,Y 601.426,Z 275.573,A -85,B 0,C 180,E1 -757.42,E2 -757.42} C_VEL
LIN {X 0,Y 601.404,Z 275.567,A -85,B 0,C 180,E1 -759.996,E2 -759.996} C_VEL
LIN {X 0,Y 601.406,Z 275.564,A -85,B 0,C 180,E1 -762.671,E2 -762.671} C_VEL
LIN {X 0,Y 601.418,Z 275.572,A -85,B 0,C 180,E1 -765.483,E2 -765.483} C_VEL
LIN {X 0,Y 601.422,Z 275.563,A -85,B 0,C 180,E1 -768.407,E2 -768.407} C_VEL
LIN {X 0,Y 601.428,Z 275.562,A -85,B 0,C 180,E1 -770.877,E2 -770.877} C_VEL
LIN {X 0,Y 601.438,Z 275.571,A -85,B 0,C 180,E1 -773.735,E2 -773.735} C_VEL
LIN {X 0,Y 601.421,Z 275.563,A -85,B 0,C 180,E1 -776.688,E2 -776.688} C_VEL
LIN {X 0,Y 601.42,Z 275.563,A -85,B 0,C 180,E1 -779.06,E2 -779.06} C_VEL
LIN {X 0,Y 601.428,Z 275.564,A -85,B 0,C 180,E1 -781.374,E2 -781.374} C_VEL
LIN {X 0,Y 601.399,Z 275.57,A -85,B 0,C 180,E1 -783.638,E2 -783.638} C_VEL
LIN {X 0,Y 601.417,Z 275.57,A -85,B 0,C 180,E1 -786.591,E2 -786.591} C_VEL
LIN {X 0,Y 601.422,Z 275.589,A -85,B 0,C 180,E1 -787.137,E2 -787.137} C_VEL
LIN {X 0,Y 601.697,Z 280.784,A -85,B 0,C 180,E1 -787.875,E2 -787.875} C_VEL
LIN {X 0,Y 601.6,Z 302.772,A -85,B 0,C 180,E1 -790.908,E2 -790.908} C_VEL
LIN {X 0,Y 601.524,Z 323.483,A -85,B 0,C 180,E1 -793.717,E2 -793.717} C_VEL
LIN {X 0,Y 601.468,Z 344.195,A -85,B 0,C 180,E1 -796.486,E2 -796.486} C_VEL
LIN {X 0,Y 601.426,Z 346.622,A -85,B 0,C 180,E1 -796.808,E2 -796.808} C_VEL
LIN {X 0,Y 601.667,Z 350.818,A -85,B 0,C 180,E1 -796.878,E2 -796.878} C_VEL
LIN {X 0,Y 601.593,Z 455.009,A -85,B 0,C 180,E1 -798.14,E2 -798.14} C_VEL
LIN {X 0,Y 601.556,Z 468.258,A -85,B 0,C 180,E1 -798.439,E2 -798.439} C_VEL
LIN {X 0,Y 601.539,Z 480.668,A -85,B 0,C 180,E1 -798.854,E2 -798.854} C_VEL
LIN {X 0,Y 601.521,Z 492.655,A -85,B 0,C 180,E1 -799.397,E2 -799.397} C_VEL
LIN {X 0,Y 601.472,Z 504.216,A -85,B 0,C 180,E1 -800.077,E2 -800.077} C_VEL
LIN {X 0,Y 601.444,Z 514.609,A -85,B 0,C 180,E1 -800.84,E2 -800.84} C_VEL
LIN {X 0,Y 601.404,Z 523.027,A -85,B 0,C 180,E1 -801.602,E2 -801.602} C_VEL
LIN {X 0,Y 601.417,Z 530.97,A -85,B 0,C 180,E1 -802.447,E2 -802.447} C_VEL
LIN {X 0,Y 601.365,Z 538.255,A -85,B 0,C 180,E1 -803.402,E2 -803.402} C_VEL
LIN {X 0,Y 601.372,Z 543.872,A -85,B 0,C 180,E1 -804.3,E2 -804.3} C_VEL
LIN {X 0,Y 601.336,Z 548.954,A -85,B 0,C 180,E1 -805.308,E2 -805.308} C_VEL
LIN {X 0,Y 601.367,Z 552.899,A -85,B 0,C 180,E1 -806.316,E2 -806.316} C_VEL
LIN {X 0,Y 601.325,Z 555.811,A -85,B 0,C 180,E1 -807.321,E2 -807.321} C_VEL
LIN {X 0,Y 601.341,Z 557.203,A -85,B 0,C 180,E1 -807.992,E2 -807.992} C_VEL
LIN {X 0,Y 601.339,Z 558.784,A -85,B 0,C 180,E1 -809.331,E2 -809.331} C_VEL
LIN {X 0,Y 601.335,Z 559,A -85,B 0,C 180,E1 -810.001,E2 -810.001} C_VEL
LIN {X 0,Y 601.347,Z 558.183,A -85,B 0,C 180,E1 -811.34,E2 -811.34} C_VEL
LIN {X 0,Y 601.341,Z 557.2,A -85,B 0,C 180,E1 -812.01,E2 -812.01} C_VEL
LIN {X 0,Y 601.325,Z 555.807,A -85,B 0,C 180,E1 -812.681,E2 -812.681} C_VEL
LIN {X 0,Y 601.367,Z 552.893,A -85,B 0,C 180,E1 -813.686,E2 -813.686} C_VEL
LIN {X 0,Y 601.336,Z 548.946,A -85,B 0,C 180,E1 -814.694,E2 -814.694} C_VEL
LIN {X 0,Y 601.372,Z 542.871,A -85,B 0,C 180,E1 -815.87,E2 -815.87} C_VEL
LIN {X 0,Y 601.382,Z 536.229,A -85,B 0,C 180,E1 -816.881,E2 -816.881} C_VEL
LIN {X 0,Y 601.401,Z 527.981,A -85,B 0,C 180,E1 -817.893,E2 -817.893} C_VEL
LIN {X 0,Y 601.435,Z 517.589,A -85,B 0,C 180,E1 -818.908,E2 -818.908} C_VEL
LIN {X 0,Y 601.46,Z 506.734,A -85,B 0,C 180,E1 -819.756,E2 -819.756} C_VEL
LIN {X 0,Y 601.494,Z 495.759,A -85,B 0,C 180,E1 -820.435,E2 -820.435} C_VEL
LIN {X 0,Y 601.549,Z 483.674,A -85,B 0,C 180,E1 -821.022,E2 -821.022} C_VEL
LIN {X 0,Y 601.531,Z 471.85,A -85,B 0,C 180,E1 -821.457,E2 -821.457} C_VEL
LIN {X 0,Y 601.578,Z 459.464,A -85,B 0,C 180,E1 -821.777,E2 -821.777} C_VEL
LIN {X 0,Y 601.608,Z 443.659,A -85,B 0,C 180,E1 -822.011,E2 -822.011} C_VEL
LIN {X 0,Y 601.479,Z 347.07,A -85,B 0,C 180,E1 -823.171,E2 -823.171} C_VEL
LIN {X 0,Y 601.436,Z 345.474,A -85,B 0,C 180,E1 -823.344,E2 -823.344} C_VEL
LIN {X 0,Y 601.467,Z 326.057,A -85,B 0,C 180,E1 -825.939,E2 -825.939} C_VEL
LIN {X 0,Y 601.575,Z 306.205,A -85,B 0,C 180,E1 -828.624,E2 -828.624} C_VEL
LIN {X 0,Y 601.655,Z 284.634,A -85,B 0,C 180,E1 -831.59,E2 -831.59} C_VEL
LIN {X 0,Y 601.632,Z 276.868,A -85,B 0,C 180,E1 -832.675,E2 -832.675} C_VEL
LIN {X 0,Y 601.418,Z 275.567,A -85,B 0,C 180,E1 -832.888,E2 -832.888} C_VEL
LIN {X 0,Y 601.399,Z 275.566,A -85,B 0,C 180,E1 -834.879,E2 -834.879} C_VEL
LIN {X 0,Y 601.413,Z 275.565,A -85,B 0,C 180,E1 -837.361,E2 -837.361} C_VEL
LIN {X 0,Y 601.434,Z 275.572,A -85,B 0,C 180,E1 -840.164,E2 -840.164} C_VEL
LIN {X 0,Y 601.422,Z 275.565,A -85,B 0,C 180,E1 -842.715,E2 -842.715} C_VEL
LIN {X 0,Y 601.392,Z 275.566,A -85,B 0,C 180,E1 -845.111,E2 -845.111} C_VEL
LIN {X 0,Y 601.438,Z 275.56,A -85,B 0,C 180,E1 -847.42,E2 -847.42} C_VEL
LIN {X 0,Y 601.404,Z 275.568,A -85,B 0,C 180,E1 -849.996,E2 -849.996} C_VEL
LIN {X 0,Y 601.412,Z 275.573,A -85,B 0,C 180,E1 -852.671,E2 -852.671} C_VEL
LIN {X 0,Y 601.404,Z 275.565,A -85,B 0,C 180,E1 -855.48,E2 -855.48} C_VEL
LIN {X 0,Y 601.423,Z 275.567,A -85,B 0,C 180,E1 -858.408,E2 -858.408} C_VEL
LIN {X 0,Y 601.409,Z 275.575,A -85,B 0,C 180,E1 -860.873,E2 -860.873} C_VEL
LIN {X 0,Y 601.406,Z 275.567,A -85,B 0,C 180,E1 -863.417,E2 -863.417} C_VEL
LIN {X 0,Y 601.421,Z 275.562,A -85,B 0,C 180,E1 -866.067,E2 -866.067} C_VEL
LIN {X 0,Y 601.421,Z 275.565,A -85,B 0,C 180,E1 -868.546,E2 -868.546} C_VEL
LIN {X 0,Y 601.431,Z 275.568,A -85,B 0,C 180,E1 -871.373,E2 -871.373} C_VEL
LIN {X 0,Y 601.411,Z 275.564,A -85,B 0,C 180,E1 -874.134,E2 -874.134} C_VEL
LIN {X 0,Y 601.397,Z 275.566,A -85,B 0,C 180,E1 -876.589,E2 -876.589} C_VEL
LIN {X 0,Y 601.432,Z 275.572,A -85,B 0,C 180,E1 -879.478,E2 -879.478} C_VEL
LIN {X 0,Y 601.391,Z 275.566,A -85,B 0,C 180,E1 -882.311,E2 -882.311} C_VEL
LIN {X 0,Y 601.409,Z 275.564,A -85,B 0,C 180,E1 -884.408,E2 -884.408} C_VEL
LIN {X 0,Y 601.415,Z 275.566,A -85,B 0,C 180,E1 -887.172,E2 -887.172} C_VEL
LIN {X 0,Y 601.428,Z 275.57,A -85,B 0,C 180,E1 -889.905,E2 -889.905} C_VEL
LIN {X 0,Y 601.443,Z 275.56,A -85,B 0,C 180,E1 -892.615,E2 -892.615} C_VEL
LIN {X 0,Y 601.411,Z 275.565,A -85,B 0,C 180,E1 -895.308,E2 -895.308} C_VEL
LIN {X 0,Y 601.436,Z 275.571,A -85,B 0,C 180,E1 -897.991,E2 -897.991} C_VEL
LIN {X 0,Y 601.446,Z 275.562,A -85,B 0,C 180,E1 -900.669,E2 -900.669} C_VEL
LIN {X 0,Y 601.429,Z 275.561,A -85,B 0,C 180,E1 -903.349,E2 -903.349} C_VEL
LIN {X 0,Y 601.401,Z 275.571,A -85,B 0,C 180,E1 -906.037,E2 -906.037} C_VEL
LIN {X 0,Y 601.418,Z 275.568,A -85,B 0,C 180,E1 -908.738,E2 -908.738} C_VEL
LIN {X 0,Y 601.435,Z 275.56,A -85,B 0,C 180,E1 -911.458,E2 -911.458} C_VEL
LIN {X 0,Y 601.406,Z 275.568,A -85,B 0,C 180,E1 -912.369,E2 -912.369} C_VEL
LIN {X 0,Y 600.744,Z 275.652,A -85,B 0,C 180,E1 -912.928,E2 -912.928} C_VEL
LIN {X 0,Y 597.897,Z 276.006,A -85,B 0,C 180,E1 -913.836,E2 -913.836} C_VEL
LIN {X 0,Y 595.486,Z 276.313,A -85,B 0,C 180,E1 -914.566,E2 -914.566} C_VEL
LIN {X 0,Y 594.446,Z 276.434,A -85,B 0,C 180,E1 -915.13,E2 -915.13} C_VEL
LIN {X 0,Y 594.359,Z 276.443,A -85,B 0,C 180,E1 -915.321,E2 -915.321} C_VEL
LIN {X 0,Y 594.389,Z 276.441,A -85,B 0,C 180,E1 -917.193,E2 -917.193} C_VEL
LIN {X 0,Y 594.371,Z 276.441,A -85,B 0,C 180,E1 -920.054,E2 -920.054} C_VEL
LIN {X 0,Y 594.361,Z 276.451,A -85,B 0,C 180,E1 -922.967,E2 -922.967} C_VEL
LIN {X 0,Y 594.376,Z 276.446,A -85,B 0,C 180,E1 -925.193,E2 -925.193} C_VEL
LIN {X 0,Y 594.39,Z 276.441,A -85,B 0,C 180,E1 -927.526,E2 -927.526} C_VEL
LIN {X 0,Y 594.389,Z 276.439,A -85,B 0,C 180,E1 -930.328,E2 -930.328} C_VEL
LIN {X 0,Y 594.379,Z 276.446,A -85,B 0,C 180,E1 -932.95,E2 -932.95} C_VEL
LIN {X 0,Y 594.35,Z 276.452,A -85,B 0,C 180,E1 -935.409,E2 -935.409} C_VEL
LIN {X 0,Y 594.386,Z 276.441,A -85,B 0,C 180,E1 -937.941,E2 -937.941} C_VEL
LIN {X 0,Y 594.375,Z 276.442,A -85,B 0,C 180,E1 -940.821,E2 -940.821} C_VEL
LIN {X 0,Y 594.369,Z 276.448,A -85,B 0,C 180,E1 -943.299,E2 -943.299} C_VEL
LIN {X 0,Y 594.363,Z 276.444,A -85,B 0,C 180,E1 -946.161,E2 -946.161} C_VEL
LIN {X 0,Y 594.382,Z 276.439,A -85,B 0,C 180,E1 -948.536,E2 -948.536} C_VEL
LIN {X 0,Y 594.375,Z 276.443,A -85,B 0,C 180,E1 -951.297,E2 -951.297} C_VEL
LIN {X 0,Y 594.352,Z 276.452,A -85,B 0,C 180,E1 -953.755,E2 -953.755} C_VEL
LIN {X 0,Y 594.378,Z 276.446,A -85,B 0,C 180,E1 -956.238,E2 -956.238} C_VEL
LIN {X 0,Y 594.371,Z 276.442,A -85,B 0,C 180,E1 -958.649,E2 -958.649} C_VEL
LIN {X 0,Y 594.384,Z 276.439,A -85,B 0,C 180,E1 -961.042,E2 -961.042} C_VEL
LIN {X 0,Y 594.388,Z 276.445,A -85,B 0,C 180,E1 -963.977,E2 -963.977} C_VEL
LIN {X 0,Y 594.388,Z 276.45,A -85,B 0,C 180,E1 -966.295,E2 -966.295} C_VEL
LIN {X 0,Y 594.405,Z 276.436,A -85,B 0,C 180,E1 -969.224,E2 -969.224} C_VEL
LIN {X 0,Y 594.346,Z 276.448,A -85,B 0,C 180,E1 -972.094,E2 -972.094} C_VEL
LIN {X 0,Y 594.361,Z 276.447,A -85,B 0,C 180,E1 -974.218,E2 -974.218} C_VEL
LIN {X 0,Y 594.374,Z 276.446,A -85,B 0,C 180,E1 -976.32,E2 -976.32} C_VEL
LIN {X 0,Y 594.376,Z 276.444,A -85,B 0,C 180,E1 -979.094,E2 -979.094} C_VEL
LIN {X 0,Y 594.382,Z 276.44,A -85,B 0,C 180,E1 -981.842,E2 -981.842} C_VEL
LIN {X 0,Y 594.39,Z 276.445,A -85,B 0,C 180,E1 -984.571,E2 -984.571} C_VEL
LIN {X 0,Y 594.415,Z 276.558,A -85,B 0,C 180,E1 -986.186,E2 -986.186} C_VEL
LIN {X 0,Y 594.455,Z 290.569,A -85,B 0,C 180,E1 -988.644,E2 -988.644} C_VEL
LIN {X 0,Y 594.353,Z 306.242,A -85,B 0,C 180,E1 -991.354,E2 -991.354} C_VEL
LIN {X 0,Y 594.363,Z 308.335,A -85,B 0,C 180,E1 -991.714,E2 -991.714} C_VEL
LIN {X 0,Y 594.755,Z 313.288,A -85,B 0,C 180,E1 -991.798,E2 -991.798} C_VEL
LIN {X 0,Y 594.589,Z 415.24,A -85,B 0,C 180,E1 -993.048,E2 -993.048} C_VEL
LIN {X 0,Y 594.59,Z 428.199,A -85,B 0,C 180,E1 -993.345,E2 -993.345} C_VEL
LIN {X 0,Y 594.6,Z 440.699,A -85,B 0,C 180,E1 -993.769,E2 -993.769} C_VEL
LIN {X 0,Y 594.498,Z 452.755,A -85,B 0,C 180,E1 -994.321,E2 -994.321} C_VEL
LIN {X 0,Y 594.425,Z 464.194,A -85,B 0,C 180,E1 -995.001,E2 -995.001} C_VEL
LIN {X 0,Y 594.433,Z 474.494,A -85,B 0,C 180,E1 -995.767,E2 -995.767} C_VEL
LIN {X 0,Y 594.382,Z 483.142,A -85,B 0,C 180,E1 -996.557,E2 -996.557} C_VEL
LIN {X 0,Y 594.339,Z 491.55,A -85,B 0,C 180,E1 -997.473,E2 -997.473} C_VEL
LIN {X 0,Y 594.303,Z 499.115,A -85,B 0,C 180,E1 -998.499,E2 -998.499} C_VEL
LIN {X 0,Y 594.271,Z 505.217,A -85,B 0,C 180,E1 -999.529,E2 -999.529} C_VEL
LIN {X 0,Y 594.289,Z 510.056,A -85,B 0,C 180,E1 -1000.561,E2 -1000.561} C_VEL
LIN {X 0,Y 594.245,Z 513.778,A -85,B 0,C 180,E1 -1001.597,E2 -1001.597} C_VEL
LIN {X 0,Y 594.238,Z 515.699,A -85,B 0,C 180,E1 -1002.29,E2 -1002.29} C_VEL
LIN {X 0,Y 594.243,Z 517.157,A -85,B 0,C 180,E1 -1002.985,E2 -1002.985} C_VEL
LIN {X 0,Y 594.257,Z 518.616,A -85,B 0,C 180,E1 -1004.123,E2 -1004.123} C_VEL
LIN {X 0,Y 594.209,Z 518.997,A -85,B 0,C 180,E1 -1005.081,E2 -1005.081} C_VEL
LIN {X 0,Y 594.222,Z 518.742,A -85,B 0,C 180,E1 -1005.784,E2 -1005.784} C_VEL
LIN {X 0,Y 594.237,Z 517.863,A -85,B 0,C 180,E1 -1006.669,E2 -1006.669} C_VEL
LIN {X 0,Y 594.215,Z 515.416,A -85,B 0,C 180,E1 -1007.908,E2 -1007.908} C_VEL
LIN {X 0,Y 594.243,Z 512.493,A -85,B 0,C 180,E1 -1008.89,E2 -1008.89} C_VEL
LIN {X 0,Y 594.261,Z 507.732,A -85,B 0,C 180,E1 -1010.056,E2 -1010.056} C_VEL
LIN {X 0,Y 594.314,Z 502.027,A -85,B 0,C 180,E1 -1011.128,E2 -1011.128} C_VEL
LIN {X 0,Y 594.313,Z 494.586,A -85,B 0,C 180,E1 -1012.234,E2 -1012.234} C_VEL
LIN {X 0,Y 594.366,Z 486.912,A -85,B 0,C 180,E1 -1013.15,E2 -1013.15} C_VEL
LIN {X 0,Y 594.395,Z 476.384,A -85,B 0,C 180,E1 -1014.166,E2 -1014.166} C_VEL
LIN {X 0,Y 594.467,Z 465.494,A -85,B 0,C 180,E1 -1015.001,E2 -1015.001} C_VEL
LIN {X 0,Y 594.494,Z 454.839,A -85,B 0,C 180,E1 -1015.655,E2 -1015.655} C_VEL
LIN {X 0,Y 594.589,Z 442.855,A -85,B 0,C 180,E1 -1016.234,E2 -1016.234} C_VEL
LIN {X 0,Y 594.599,Z 430.224,A -85,B 0,C 180,E1 -1016.688,E2 -1016.688} C_VEL
LIN {X 0,Y 594.637,Z 417.09,A -85,B 0,C 180,E1 -1017.006,E2 -1017.006} C_VEL
LIN {X 0,Y 594.708,Z 395.214,A -85,B 0,C 180,E1 -1017.3,E2 -1017.3} C_VEL
LIN {X 0,Y 594.63,Z 310.222,A -85,B 0,C 180,E1 -1018.332,E2 -1018.332} C_VEL
LIN {X 0,Y 594.347,Z 308.329,A -85,B 0,C 180,E1 -1018.377,E2 -1018.377} C_VEL
LIN {X 0,Y 594.44,Z 292.292,A -85,B 0,C 180,E1 -1021.146,E2 -1021.146} C_VEL
LIN {X 0,Y 594.427,Z 277.393,A -85,B 0,C 180,E1 -1023.756,E2 -1023.756} C_VEL
LIN {X 0,Y 594.317,Z 276.451,A -85,B 0,C 180,E1 -1023.944,E2 -1023.944} C_VEL
LIN {X 0,Y 594.36,Z 276.452,A -85,B 0,C 180,E1 -1027.087,E2 -1027.087} C_VEL
LIN {X 0,Y 594.318,Z 276.451,A -85,B 0,C 180,E1 -1029.768,E2 -1029.768} C_VEL
LIN {X 0,Y 594.309,Z 276.449,A -85,B 0,C 180,E1 -1032.379,E2 -1032.379} C_VEL
LIN {X 0,Y 594.315,Z 276.455,A -85,B 0,C 180,E1 -1035.194,E2 -1035.194} C_VEL
LIN {X 0,Y 594.351,Z 276.445,A -85,B 0,C 180,E1 -1038.153,E2 -1038.153} C_VEL
LIN {X 0,Y 594.339,Z 276.445,A -85,B 0,C 180,E1 -1040.317,E2 -1040.317} C_VEL
LIN {X 0,Y 594.311,Z 276.45,A -85,B 0,C 180,E1 -1042.908,E2 -1042.908} C_VEL
LIN {X 0,Y 594.354,Z 276.451,A -85,B 0,C 180,E1 -1045.863,E2 -1045.863} C_VEL
LIN {X 0,Y 594.345,Z 276.444,A -85,B 0,C 180,E1 -1048.648,E2 -1048.648} C_VEL
LIN {X 0,Y 594.359,Z 276.443,A -85,B 0,C 180,E1 -1051.043,E2 -1051.043} C_VEL
LIN {X 0,Y 594.356,Z 276.45,A -85,B 0,C 180,E1 -1054.055,E2 -1054.055} C_VEL
LIN {X 0,Y 594.366,Z 276.446,A -85,B 0,C 180,E1 -1056.295,E2 -1056.295} C_VEL
LIN {X 0,Y 594.369,Z 276.441,A -85,B 0,C 180,E1 -1059.223,E2 -1059.223} C_VEL
LIN {X 0,Y 594.358,Z 276.453,A -85,B 0,C 180,E1 -1062.095,E2 -1062.095} C_VEL
LIN {X 0,Y 594.336,Z 276.446,A -85,B 0,C 180,E1 -1064.921,E2 -1064.921} C_VEL
LIN {X 0,Y 594.369,Z 276.444,A -85,B 0,C 180,E1 -1067.711,E2 -1067.711} C_VEL
LIN {X 0,Y 594.363,Z 276.449,A -85,B 0,C 180,E1 -1070.471,E2 -1070.471} C_VEL
LIN {X 0,Y 594.39,Z 276.445,A -85,B 0,C 180,E1 -1072.527,E2 -1072.527} C_VEL
LIN {X 0,Y 594.364,Z 276.442,A -85,B 0,C 180,E1 -1075.252,E2 -1075.252} C_VEL
LIN {X 0,Y 594.368,Z 276.444,A -85,B 0,C 180,E1 -1077.967,E2 -1077.967} C_VEL
LIN {X 0,Y 594.421,Z 276.443,A -85,B 0,C 180,E1 -1080.678,E2 -1080.678} C_VEL
LIN {X 0,Y 594.369,Z 276.44,A -85,B 0,C 180,E1 -1083.39,E2 -1083.39} C_VEL
LIN {X 0,Y 594.382,Z 276.44,A -85,B 0,C 180,E1 -1085.428,E2 -1085.428} C_VEL
LIN {X 0,Y 594.397,Z 276.44,A -85,B 0,C 180,E1 -1088.157,E2 -1088.157} C_VEL
LIN {X 0,Y 594.383,Z 276.445,A -85,B 0,C 180,E1 -1091.079,E2 -1091.079} C_VEL
LIN {X 0,Y 594.37,Z 276.44,A -85,B 0,C 180,E1 -1093.679,E2 -1093.679} C_VEL
LIN {X 0,Y 594.376,Z 276.448,A -85,B 0,C 180,E1 -1096.719,E2 -1096.719} C_VEL
LIN {X 0,Y 594.357,Z 276.447,A -85,B 0,C 180,E1 -1099.335,E2 -1099.335} C_VEL
LIN {X 0,Y 594.354,Z 276.446,A -85,B 0,C 180,E1 -1101.504,E2 -1101.504} C_VEL
LIN {X 0,Y 594.376,Z 276.441,A -85,B 0,C 180,E1 -1104.447,E2 -1104.447} C_VEL
LIN {X 0,Y 594.378,Z 276.444,A -85,B 0,C 180,E1 -1106.7,E2 -1106.7} C_VEL
LIN {X 0,Y 594.369,Z 276.448,A -85,B 0,C 180,E1 -1108.999,E2 -1108.999} C_VEL
LIN {X 0,Y 594.383,Z 276.443,A -85,B 0,C 180,E1 -1111.646,E2 -1111.646} C_VEL
LIN {X 0,Y 594.382,Z 276.44,A -85,B 0,C 180,E1 -1114.58,E2 -1114.58} C_VEL
LIN {X 0,Y 594.375,Z 276.446,A -85,B 0,C 180,E1 -1117.088,E2 -1117.088} C_VEL
LIN {X 0,Y 594.367,Z 276.447,A -85,B 0,C 180,E1 -1119.776,E2 -1119.776} C_VEL
LIN {X 0,Y 594.365,Z 276.442,A -85,B 0,C 180,E1 -1122.376,E2 -1122.376} C_VEL
LIN {X 0,Y 594.355,Z 276.447,A -85,B 0,C 180,E1 -1125.192,E2 -1125.192} C_VEL
LIN {X 0,Y 594.367,Z 276.452,A -85,B 0,C 180,E1 -1127.626,E2 -1127.626} C_VEL
LIN {X 0,Y 594.384,Z 276.441,A -85,B 0,C 180,E1 -1130.322,E2 -1130.322} C_VEL
LIN {X 0,Y 594.381,Z 276.44,A -85,B 0,C 180,E1 -1132.915,E2 -1132.915} C_VEL
LIN {X 0,Y 594.376,Z 276.451,A -85,B 0,C 180,E1 -1135.863,E2 -1135.863} C_VEL
LIN {X 0,Y 594.368,Z 276.442,A -85,B 0,C 180,E1 -1138.651,E2 -1138.651} C_VEL
LIN {X 0,Y 594.379,Z 276.44,A -85,B 0,C 180,E1 -1141.043,E2 -1141.043} C_VEL
LIN {X 0,Y 594.381,Z 276.451,A -85,B 0,C 180,E1 -1143.979,E2 -1143.979} C_VEL
LIN {X 0,Y 594.384,Z 276.446,A -85,B 0,C 180,E1 -1146.667,E2 -1146.667} C_VEL
LIN {X 0,Y 594.419,Z 276.559,A -85,B 0,C 180,E1 -1146.99,E2 -1146.99} C_VEL
LIN {X 0,Y 594.773,Z 283.355,A -85,B 0,C 180,E1 -1147.967,E2 -1147.967} C_VEL
LIN {X 0,Y 594.616,Z 305.987,A -85,B 0,C 180,E1 -1151.12,E2 -1151.12} C_VEL
LIN {X 0,Y 594.498,Z 326.072,A -85,B 0,C 180,E1 -1153.872,E2 -1153.872} C_VEL
LIN {X 0,Y 594.439,Z 345.489,A -85,B 0,C 180,E1 -1156.498,E2 -1156.498} C_VEL
LIN {X 0,Y 594.441,Z 346.622,A -85,B 0,C 180,E1 -1156.65,E2 -1156.65} C_VEL
LIN {X 0,Y 594.776,Z 350.818,A -85,B 0,C 180,E1 -1156.723,E2 -1156.723} C_VEL
LIN {X 0,Y 594.645,Z 455.009,A -85,B 0,C 180,E1 -1158,E2 -1158} C_VEL
LIN {X 0,Y 594.62,Z 468.259,A -85,B 0,C 180,E1 -1158.302,E2 -1158.302} C_VEL
LIN {X 0,Y 594.593,Z 480.461,A -85,B 0,C 180,E1 -1158.714,E2 -1158.714} C_VEL
LIN {X 0,Y 594.533,Z 492.653,A -85,B 0,C 180,E1 -1159.271,E2 -1159.271} C_VEL
LIN {X 0,Y 594.46,Z 504.217,A -85,B 0,C 180,E1 -1159.958,E2 -1159.958} C_VEL
LIN {X 0,Y 594.413,Z 514.611,A -85,B 0,C 180,E1 -1160.731,E2 -1160.731} C_VEL
LIN {X 0,Y 594.349,Z 523.04,A -85,B 0,C 180,E1 -1161.501,E2 -1161.501} C_VEL
LIN {X 0,Y 594.346,Z 530.97,A -85,B 0,C 180,E1 -1162.356,E2 -1162.356} C_VEL
LIN {X 0,Y 594.28,Z 538.83,A -85,B 0,C 180,E1 -1163.411,E2 -1163.411} C_VEL
LIN {X 0,Y 594.289,Z 545.686,A -85,B 0,C 180,E1 -1164.572,E2 -1164.572} C_VEL
LIN {X 0,Y 594.27,Z 550.376,A -85,B 0,C 180,E1 -1165.592,E2 -1165.592} C_VEL
LIN {X 0,Y 594.267,Z 553.96,A -85,B 0,C 180,E1 -1166.611,E2 -1166.611} C_VEL
LIN {X 0,Y 594.225,Z 555.811,A -85,B 0,C 180,E1 -1167.289,E2 -1167.289} C_VEL
LIN {X 0,Y 594.24,Z 557.203,A -85,B 0,C 180,E1 -1167.968,E2 -1167.968} C_VEL
LIN {X 0,Y 594.239,Z 558.785,A -85,B 0,C 180,E1 -1169.323,E2 -1169.323} C_VEL
LIN {X 0,Y 594.236,Z 559,A -85,B 0,C 180,E1 -1170.001,E2 -1170.001} C_VEL
LIN {X 0,Y 594.247,Z 558.184,A -85,B 0,C 180,E1 -1171.356,E2 -1171.356} C_VEL
LIN {X 0,Y 594.24,Z 557.2,A -85,B 0,C 180,E1 -1172.034,E2 -1172.034} C_VEL
LIN {X 0,Y 594.226,Z 555.807,A -85,B 0,C 180,E1 -1172.713,E2 -1172.713} C_VEL
LIN {X 0,Y 594.289,Z 552.893,A -85,B 0,C 180,E1 -1173.73,E2 -1173.73} C_VEL
LIN {X 0,Y 594.241,Z 548.946,A -85,B 0,C 180,E1 -1174.75,E2 -1174.75} C_VEL
LIN {X 0,Y 594.304,Z 542.872,A -85,B 0,C 180,E1 -1175.94,E2 -1175.94} C_VEL
LIN {X 0,Y 594.309,Z 536.229,A -85,B 0,C 180,E1 -1176.963,E2 -1176.963} C_VEL
LIN {X 0,Y 594.36,Z 527.982,A -85,B 0,C 180,E1 -1177.987,E2 -1177.987} C_VEL
LIN {X 0,Y 594.404,Z 517.59,A -85,B 0,C 180,E1 -1179.014,E2 -1179.014} C_VEL
LIN {X 0,Y 594.448,Z 506.734,A -85,B 0,C 180,E1 -1179.872,E2 -1179.872} C_VEL
LIN {X 0,Y 594.506,Z 495.761,A -85,B 0,C 180,E1 -1180.559,E2 -1180.559} C_VEL
LIN {X 0,Y 594.566,Z 483.555,A -85,B 0,C 180,E1 -1181.159,E2 -1181.159} C_VEL
LIN {X 0,Y 594.576,Z 471.848,A -85,B 0,C 180,E1 -1181.593,E2 -1181.593} C_VEL
LIN {X 0,Y 594.634,Z 459.463,A -85,B 0,C 180,E1 -1181.916,E2 -1181.916} C_VEL
LIN {X 0,Y 594.69,Z 443.659,A -85,B 0,C 180,E1 -1182.153,E2 -1182.153} C_VEL
LIN {X 0,Y 594.623,Z 348.189,A -85,B 0,C 180,E1 -1183.312,E2 -1183.312} C_VEL
LIN {X 0,Y 594.442,Z 346.606,A -85,B 0,C 180,E1 -1183.352,E2 -1183.352} C_VEL
LIN {X 0,Y 594.499,Z 326.057,A -85,B 0,C 180,E1 -1186.13,E2 -1186.13} C_VEL
LIN {X 0,Y 594.608,Z 306.004,A -85,B 0,C 180,E1 -1188.878,E2 -1188.878} C_VEL
LIN {X 0,Y 594.731,Z 284.634,A -85,B 0,C 180,E1 -1191.855,E2 -1191.855} C_VEL
LIN {X 0,Y 594.669,Z 277.933,A -85,B 0,C 180,E1 -1192.804,E2 -1192.804} C_VEL
LIN {X 0,Y 594.391,Z 276.444,A -85,B 0,C 180,E1 -1193.059,E2 -1193.059} C_VEL
LIN {X 0,Y 594.365,Z 276.443,A -85,B 0,C 180,E1 -1195.194,E2 -1195.194} C_VEL
LIN {X 0,Y 594.374,Z 276.443,A -85,B 0,C 180,E1 -1197.524,E2 -1197.524} C_VEL
LIN {X 0,Y 594.391,Z 276.446,A -85,B 0,C 180,E1 -1200.328,E2 -1200.328} C_VEL
LIN {X 0,Y 594.381,Z 276.44,A -85,B 0,C 180,E1 -1202.951,E2 -1202.951} C_VEL
LIN {X 0,Y 594.351,Z 276.443,A -85,B 0,C 180,E1 -1205.41,E2 -1205.41} C_VEL
LIN {X 0,Y 594.383,Z 276.443,A -85,B 0,C 180,E1 -1207.942,E2 -1207.942} C_VEL
LIN {X 0,Y 594.378,Z 276.445,A -85,B 0,C 180,E1 -1210.822,E2 -1210.822} C_VEL
LIN {X 0,Y 594.37,Z 276.441,A -85,B 0,C 180,E1 -1213.3,E2 -1213.3} C_VEL
LIN {X 0,Y 594.365,Z 276.444,A -85,B 0,C 180,E1 -1216.162,E2 -1216.162} C_VEL
LIN {X 0,Y 594.381,Z 276.447,A -85,B 0,C 180,E1 -1218.536,E2 -1218.536} C_VEL
LIN {X 0,Y 594.378,Z 276.443,A -85,B 0,C 180,E1 -1221.297,E2 -1221.297} C_VEL
LIN {X 0,Y 594.355,Z 276.443,A -85,B 0,C 180,E1 -1223.755,E2 -1223.755} C_VEL
LIN {X 0,Y 594.368,Z 276.441,A -85,B 0,C 180,E1 -1226.238,E2 -1226.238} C_VEL
LIN {X 0,Y 594.372,Z 276.444,A -85,B 0,C 180,E1 -1228.65,E2 -1228.65} C_VEL
LIN {X 0,Y 594.386,Z 276.448,A -85,B 0,C 180,E1 -1231.043,E2 -1231.043} C_VEL
LIN {X 0,Y 594.386,Z 276.439,A -85,B 0,C 180,E1 -1233.978,E2 -1233.978} C_VEL
LIN {X 0,Y 594.377,Z 276.44,A -85,B 0,C 180,E1 -1236.295,E2 -1236.295} C_VEL
LIN {X 0,Y 594.406,Z 276.444,A -85,B 0,C 180,E1 -1239.224,E2 -1239.224} C_VEL
LIN {X 0,Y 594.351,Z 276.445,A -85,B 0,C 180,E1 -1242.095,E2 -1242.095} C_VEL
LIN {X 0,Y 594.364,Z 276.443,A -85,B 0,C 180,E1 -1244.219,E2 -1244.219} C_VEL
LIN {X 0,Y 594.379,Z 276.441,A -85,B 0,C 180,E1 -1246.321,E2 -1246.321} C_VEL
LIN {X 0,Y 594.37,Z 276.442,A -85,B 0,C 180,E1 -1249.094,E2 -1249.094} C_VEL
LIN {X 0,Y 594.384,Z 276.451,A -85,B 0,C 180,E1 -1251.843,E2 -1251.843} C_VEL
LIN {X 0,Y 594.395,Z 276.439,A -85,B 0,C 180,E1 -1254.572,E2 -1254.572} C_VEL
LIN {X 0,Y 594.399,Z 276.438,A -85,B 0,C 180,E1 -1257.289,E2 -1257.289} C_VEL
LIN {X 0,Y 594.413,Z 276.445,A -85,B 0,C 180,E1 -1260,E2 -1260} C_VEL
LIN {X 0,Y 594.405,Z 276.439,A -85,B 0,C 180,E1 -1262.711,E2 -1262.711} C_VEL
LIN {X 0,Y 594.392,Z 276.438,A -85,B 0,C 180,E1 -1265.428,E2 -1265.428} C_VEL
LIN {X 0,Y 594.381,Z 276.447,A -85,B 0,C 180,E1 -1268.157,E2 -1268.157} C_VEL
LIN {X 0,Y 594.393,Z 276.439,A -85,B 0,C 180,E1 -1271.073,E2 -1271.073} C_VEL
LIN {X 0,Y 594.374,Z 276.44,A -85,B 0,C 180,E1 -1273.679,E2 -1273.679} C_VEL
LIN {X 0,Y 594.359,Z 276.443,A -85,B 0,C 180,E1 -1275.321,E2 -1275.321} C_VEL
LIN {X 0,Y 593.681,Z 276.528,A -85,B 0,C 180,E1 -1275.887,E2 -1275.887} C_VEL
LIN {X 0,Y 590.809,Z 276.893,A -85,B 0,C 180,E1 -1276.805,E2 -1276.805} C_VEL
LIN {X 0,Y 588.399,Z 277.189,A -85,B 0,C 180,E1 -1277.543,E2 -1277.543} C_VEL
LIN {X 0,Y 587.379,Z 277.314,A -85,B 0,C 180,E1 -1278.113,E2 -1278.113} C_VEL
LIN {X 0,Y 587.304,Z 277.324,A -85,B 0,C 180,E1 -1278.306,E2 -1278.306} C_VEL
LIN {X 0,Y 587.335,Z 277.324,A -85,B 0,C 180,E1 -1281.037,E2 -1281.037} C_VEL
LIN {X 0,Y 587.317,Z 277.324,A -85,B 0,C 180,E1 -1283.259,E2 -1283.259} C_VEL
LIN {X 0,Y 587.335,Z 277.319,A -85,B 0,C 180,E1 -1285.517,E2 -1285.517} C_VEL
LIN {X 0,Y 587.349,Z 277.316,A -85,B 0,C 180,E1 -1287.818,E2 -1287.818} C_VEL
LIN {X 0,Y 587.339,Z 277.318,A -85,B 0,C 180,E1 -1290.509,E2 -1290.509} C_VEL
LIN {X 0,Y 587.335,Z 277.325,A -85,B 0,C 180,E1 -1293.397,E2 -1293.397} C_VEL
LIN {X 0,Y 587.292,Z 277.324,A -85,B 0,C 180,E1 -1295.9,E2 -1295.9} C_VEL
LIN {X 0,Y 587.324,Z 277.318,A -85,B 0,C 180,E1 -1298.48,E2 -1298.48} C_VEL
LIN {X 0,Y 587.338,Z 277.322,A -85,B 0,C 180,E1 -1301.157,E2 -1301.157} C_VEL
LIN {X 0,Y 587.315,Z 277.322,A -85,B 0,C 180,E1 -1304.111,E2 -1304.111} C_VEL
LIN {X 0,Y 587.317,Z 277.321,A -85,B 0,C 180,E1 -1306.993,E2 -1306.993} C_VEL
LIN {X 0,Y 587.313,Z 277.331,A -85,B 0,C 180,E1 -1309.745,E2 -1309.745} C_VEL
LIN {X 0,Y 587.348,Z 277.318,A -85,B 0,C 180,E1 -1312.392,E2 -1312.392} C_VEL
LIN {X 0,Y 587.361,Z 277.322,A -85,B 0,C 180,E1 -1315.779,E2 -1315.779} C_VEL
LIN {X 0,Y 587.34,Z 277.324,A -85,B 0,C 180,E1 -1318.23,E2 -1318.23} C_VEL
LIN {X 0,Y 587.352,Z 277.315,A -85,B 0,C 180,E1 -1320.866,E2 -1320.866} C_VEL
LIN {X 0,Y 587.362,Z 277.318,A -85,B 0,C 180,E1 -1323.818,E2 -1323.818} C_VEL
LIN {X 0,Y 587.328,Z 277.324,A -85,B 0,C 180,E1 -1325.992,E2 -1325.992} C_VEL
LIN {X 0,Y 587.321,Z 277.328,A -85,B 0,C 180,E1 -1328.225,E2 -1328.225} C_VEL
LIN {X 0,Y 587.351,Z 277.316,A -85,B 0,C 180,E1 -1331.15,E2 -1331.15} C_VEL
LIN {X 0,Y 587.32,Z 277.322,A -85,B 0,C 180,E1 -1334.024,E2 -1334.024} C_VEL
LIN {X 0,Y 587.352,Z 277.318,A -85,B 0,C 180,E1 -1336.153,E2 -1336.153} C_VEL
LIN {X 0,Y 587.342,Z 277.323,A -85,B 0,C 180,E1 -1338.962,E2 -1338.962} C_VEL
LIN {X 0,Y 587.343,Z 277.317,A -85,B 0,C 180,E1 -1341.743,E2 -1341.743} C_VEL
LIN {X 0,Y 587.355,Z 277.32,A -85,B 0,C 180,E1 -1344.506,E2 -1344.506} C_VEL
LIN {X 0,Y 587.344,Z 277.378,A -85,B 0,C 180,E1 -1346.097,E2 -1346.097} C_VEL
LIN {X 0,Y 587.443,Z 285.8,A -85,B 0,C 180,E1 -1347.599,E2 -1347.599} C_VEL
LIN {X 0,Y 587.377,Z 301.392,A -85,B 0,C 180,E1 -1350.342,E2 -1350.342} C_VEL
LIN {X 0,Y 587.325,Z 308.403,A -85,B 0,C 180,E1 -1351.563,E2 -1351.563} C_VEL
LIN {X 0,Y 587.877,Z 312.164,A -85,B 0,C 180,E1 -1351.626,E2 -1351.626} C_VEL
LIN {X 0,Y 587.648,Z 415.675,A -85,B 0,C 180,E1 -1352.912,E2 -1352.912} C_VEL
LIN {X 0,Y 587.651,Z 429.224,A -85,B 0,C 180,E1 -1353.234,E2 -1353.234} C_VEL
LIN {X 0,Y 587.616,Z 442.003,A -85,B 0,C 180,E1 -1353.685,E2 -1353.685} C_VEL
LIN {X 0,Y 587.52,Z 452.908,A -85,B 0,C 180,E1 -1354.201,E2 -1354.201} C_VEL
LIN {X 0,Y 587.401,Z 464.331,A -85,B 0,C 180,E1 -1354.889,E2 -1354.889} C_VEL
LIN {X 0,Y 587.399,Z 474.607,A -85,B 0,C 180,E1 -1355.664,E2 -1355.664} C_VEL
LIN {X 0,Y 587.347,Z 483.293,A -85,B 0,C 180,E1 -1356.468,E2 -1356.468} C_VEL
LIN {X 0,Y 587.273,Z 491.622,A -85,B 0,C 180,E1 -1357.39,E2 -1357.39} C_VEL
LIN {X 0,Y 587.213,Z 499.177,A -85,B 0,C 180,E1 -1358.43,E2 -1358.43} C_VEL
LIN {X 0,Y 587.199,Z 506.174,A -85,B 0,C 180,E1 -1359.645,E2 -1359.645} C_VEL
LIN {X 0,Y 587.188,Z 510.811,A -85,B 0,C 180,E1 -1360.69,E2 -1360.69} C_VEL
LIN {X 0,Y 587.161,Z 514.343,A -85,B 0,C 180,E1 -1361.739,E2 -1361.739} C_VEL
LIN {X 0,Y 587.159,Z 516.116,A -85,B 0,C 180,E1 -1362.441,E2 -1362.441} C_VEL
LIN {X 0,Y 587.144,Z 517.455,A -85,B 0,C 180,E1 -1363.144,E2 -1363.144} C_VEL
LIN {X 0,Y 587.155,Z 518.663,A -85,B 0,C 180,E1 -1364.179,E2 -1364.179} C_VEL
LIN {X 0,Y 587.123,Z 518.956,A -85,B 0,C 180,E1 -1365.267,E2 -1365.267} C_VEL
LIN {X 0,Y 587.137,Z 518.615,A -85,B 0,C 180,E1 -1365.979,E2 -1365.979} C_VEL
LIN {X 0,Y 587.14,Z 517.774,A -85,B 0,C 180,E1 -1366.746,E2 -1366.746} C_VEL
LIN {X 0,Y 587.132,Z 516.613,A -85,B 0,C 180,E1 -1367.411,E2 -1367.411} C_VEL
LIN {X 0,Y 587.162,Z 513.908,A -85,B 0,C 180,E1 -1368.492,E2 -1368.492} C_VEL
LIN {X 0,Y 587.166,Z 510.071,A -85,B 0,C 180,E1 -1369.58,E2 -1369.58} C_VEL
LIN {X 0,Y 587.183,Z 505.065,A -85,B 0,C 180,E1 -1370.657,E2 -1370.657} C_VEL
LIN {X 0,Y 587.225,Z 498.421,A -85,B 0,C 180,E1 -1371.777,E2 -1371.777} C_VEL
LIN {X 0,Y 587.26,Z 491.701,A -85,B 0,C 180,E1 -1372.69,E2 -1372.69} C_VEL
LIN {X 0,Y 587.331,Z 483.208,A -85,B 0,C 180,E1 -1373.631,E2 -1373.631} C_VEL
LIN {X 0,Y 587.398,Z 474.617,A -85,B 0,C 180,E1 -1374.426,E2 -1374.426} C_VEL
LIN {X 0,Y 587.466,Z 463.966,A -85,B 0,C 180,E1 -1375.225,E2 -1375.225} C_VEL
LIN {X 0,Y 587.521,Z 452.954,A -85,B 0,C 180,E1 -1375.887,E2 -1375.887} C_VEL
LIN {X 0,Y 587.613,Z 440.757,A -85,B 0,C 180,E1 -1376.455,E2 -1376.455} C_VEL
LIN {X 0,Y 587.661,Z 428.246,A -85,B 0,C 180,E1 -1376.884,E2 -1376.884} C_VEL
LIN {X 0,Y 587.733,Z 414.775,A -85,B 0,C 180,E1 -1377.193,E2 -1377.193} C_VEL
LIN {X 0,Y 587.671,Z 310.854,A -85,B 0,C 180,E1 -1378.485,E2 -1378.485} C_VEL
LIN {X 0,Y 587.324,Z 308.29,A -85,B 0,C 180,E1 -1378.547,E2 -1378.547} C_VEL
LIN {X 0,Y 587.407,Z 292.198,A -85,B 0,C 180,E1 -1381.361,E2 -1381.361} C_VEL
LIN {X 0,Y 587.419,Z 278.44,A -85,B 0,C 180,E1 -1383.801,E2 -1383.801} C_VEL
LIN {X 0,Y 587.268,Z 277.33,A -85,B 0,C 180,E1 -1384.017,E2 -1384.017} C_VEL
LIN {X 0,Y 587.3,Z 277.326,A -85,B 0,C 180,E1 -1386.749,E2 -1386.749} C_VEL
LIN {X 0,Y 587.291,Z 277.333,A -85,B 0,C 180,E1 -1389.362,E2 -1389.362} C_VEL
LIN {X 0,Y 587.278,Z 277.326,A -85,B 0,C 180,E1 -1392.102,E2 -1392.102} C_VEL
LIN {X 0,Y 587.263,Z 277.332,A -85,B 0,C 180,E1 -1395.084,E2 -1395.084} C_VEL
LIN {X 0,Y 587.302,Z 277.325,A -85,B 0,C 180,E1 -1397.923,E2 -1397.923} C_VEL
LIN {X 0,Y 587.301,Z 277.322,A -85,B 0,C 180,E1 -1400.637,E2 -1400.637} C_VEL
LIN {X 0,Y 587.295,Z 277.328,A -85,B 0,C 180,E1 -1403.297,E2 -1403.297} C_VEL
LIN {X 0,Y 587.333,Z 277.327,A -85,B 0,C 180,E1 -1405.778,E2 -1405.778} C_VEL
LIN {X 0,Y 587.322,Z 277.321,A -85,B 0,C 180,E1 -1408.23,E2 -1408.23} C_VEL
LIN {X 0,Y 587.328,Z 277.318,A -85,B 0,C 180,E1 -1410.867,E2 -1410.867} C_VEL
LIN {X 0,Y 587.294,Z 277.333,A -85,B 0,C 180,E1 -1413.828,E2 -1413.828} C_VEL
LIN {X 0,Y 587.318,Z 277.33,A -85,B 0,C 180,E1 -1415.993,E2 -1415.993} C_VEL
LIN {X 0,Y 587.315,Z 277.319,A -85,B 0,C 180,E1 -1418.962,E2 -1418.962} C_VEL
LIN {X 0,Y 587.301,Z 277.329,A -85,B 0,C 180,E1 -1421.873,E2 -1421.873} C_VEL
LIN {X 0,Y 587.3,Z 277.323,A -85,B 0,C 180,E1 -1424.736,E2 -1424.736} C_VEL
LIN {X 0,Y 587.293,Z 277.323,A -85,B 0,C 180,E1 -1426.858,E2 -1426.858} C_VEL
LIN {X 0,Y 587.319,Z 277.321,A -85,B 0,C 180,E1 -1429.66,E2 -1429.66} C_VEL
LIN {X 0,Y 587.358,Z 277.322,A -85,B 0,C 180,E1 -1432.437,E2 -1432.437} C_VEL
LIN {X 0,Y 587.338,Z 277.317,A -85,B 0,C 180,E1 -1435.195,E2 -1435.195} C_VEL
LIN {X 0,Y 587.339,Z 277.319,A -85,B 0,C 180,E1 -1437.943,E2 -1437.943} C_VEL
LIN {X 0,Y 587.39,Z 277.318,A -85,B 0,C 180,E1 -1440.686,E2 -1440.686} C_VEL
LIN {X 0,Y 587.32,Z 277.318,A -85,B 0,C 180,E1 -1443.43,E2 -1443.43} C_VEL
LIN {X 0,Y 587.345,Z 277.316,A -85,B 0,C 180,E1 -1445.493,E2 -1445.493} C_VEL
LIN {X 0,Y 587.353,Z 277.318,A -85,B 0,C 180,E1 -1448.256,E2 -1448.256} C_VEL
LIN {X 0,Y 587.348,Z 277.32,A -85,B 0,C 180,E1 -1451.142,E2 -1451.142} C_VEL
LIN {X 0,Y 587.35,Z 277.316,A -85,B 0,C 180,E1 -1454.261,E2 -1454.261} C_VEL
LIN {X 0,Y 587.338,Z 277.319,A -85,B 0,C 180,E1 -1457.406,E2 -1457.406} C_VEL
LIN {X 0,Y 587.315,Z 277.321,A -85,B 0,C 180,E1 -1460.306,E2 -1460.306} C_VEL
LIN {X 0,Y 587.312,Z 277.327,A -85,B 0,C 180,E1 -1463.259,E2 -1463.259} C_VEL
LIN {X 0,Y 587.329,Z 277.322,A -85,B 0,C 180,E1 -1465.517,E2 -1465.517} C_VEL
LIN {X 0,Y 587.336,Z 277.318,A -85,B 0,C 180,E1 -1467.819,E2 -1467.819} C_VEL
LIN {X 0,Y 587.34,Z 277.318,A -85,B 0,C 180,E1 -1470.513,E2 -1470.513} C_VEL
LIN {X 0,Y 587.328,Z 277.328,A -85,B 0,C 180,E1 -1473.397,E2 -1473.397} C_VEL
LIN {X 0,Y 587.346,Z 277.318,A -85,B 0,C 180,E1 -1475.896,E2 -1475.896} C_VEL
LIN {X 0,Y 587.324,Z 277.319,A -85,B 0,C 180,E1 -1478.48,E2 -1478.48} C_VEL
LIN {X 0,Y 587.329,Z 277.324,A -85,B 0,C 180,E1 -1481.158,E2 -1481.158} C_VEL
LIN {X 0,Y 587.326,Z 277.321,A -85,B 0,C 180,E1 -1484.115,E2 -1484.115} C_VEL
LIN {X 0,Y 587.316,Z 277.321,A -85,B 0,C 180,E1 -1486.996,E2 -1486.996} C_VEL
LIN {X 0,Y 587.313,Z 277.33,A -85,B 0,C 180,E1 -1489.748,E2 -1489.748} C_VEL
LIN {X 0,Y 587.341,Z 277.318,A -85,B 0,C 180,E1 -1492.394,E2 -1492.394} C_VEL
LIN {X 0,Y 587.322,Z 277.32,A -85,B 0,C 180,E1 -1494.946,E2 -1494.946} C_VEL
LIN {X 0,Y 587.333,Z 277.321,A -85,B 0,C 180,E1 -1497.422,E2 -1497.422} C_VEL
LIN {X 0,Y 587.331,Z 277.327,A -85,B 0,C 180,E1 -1499.831,E2 -1499.831} C_VEL
LIN {X 0,Y 587.349,Z 277.322,A -85,B 0,C 180,E1 -1502.308,E2 -1502.308} C_VEL
LIN {X 0,Y 587.349,Z 277.318,A -85,B 0,C 180,E1 -1505.243,E2 -1505.243} C_VEL
LIN {X 0,Y 587.354,Z 277.427,A -85,B 0,C 180,E1 -1506.822,E2 -1506.822} C_VEL
LIN {X 0,Y 587.857,Z 280.92,A -85,B 0,C 180,E1 -1507.345,E2 -1507.345} C_VEL
LIN {X 0,Y 587.706,Z 301.478,A -85,B 0,C 180,E1 -1510.257,E2 -1510.257} C_VEL
LIN {X 0,Y 587.547,Z 320.618,A -85,B 0,C 180,E1 -1512.922,E2 -1512.922} C_VEL
LIN {X 0,Y 587.444,Z 343.04,A -85,B 0,C 180,E1 -1516,E2 -1516} C_VEL
LIN {X 0,Y 587.392,Z 346.622,A -85,B 0,C 180,E1 -1516.487,E2 -1516.487} C_VEL
LIN {X 0,Y 587.869,Z 350.818,A -85,B 0,C 180,E1 -1516.564,E2 -1516.564} C_VEL
LIN {X 0,Y 587.724,Z 455.009,A -85,B 0,C 180,E1 -1517.856,E2 -1517.856} C_VEL
LIN {X 0,Y 587.67,Z 468.26,A -85,B 0,C 180,E1 -1518.162,E2 -1518.162} C_VEL
LIN {X 0,Y 587.625,Z 480.631,A -85,B 0,C 180,E1 -1518.585,E2 -1518.585} C_VEL
LIN {X 0,Y 587.549,Z 492.652,A -85,B 0,C 180,E1 -1519.142,E2 -1519.142} C_VEL
LIN {X 0,Y 587.442,Z 504.219,A -85,B 0,C 180,E1 -1519.837,E2 -1519.837} C_VEL
LIN {X 0,Y 587.392,Z 514.612,A -85,B 0,C 180,E1 -1520.619,E2 -1520.619} C_VEL
LIN {X 0,Y 587.298,Z 523.054,A -85,B 0,C 180,E1 -1521.398,E2 -1521.398} C_VEL
LIN {X 0,Y 587.273,Z 530.97,A -85,B 0,C 180,E1 -1522.264,E2 -1522.264} C_VEL
LIN {X 0,Y 587.229,Z 537.477,A -85,B 0,C 180,E1 -1523.127,E2 -1523.127} C_VEL
LIN {X 0,Y 587.236,Z 543.872,A -85,B 0,C 180,E1 -1524.162,E2 -1524.162} C_VEL
LIN {X 0,Y 587.147,Z 548.954,A -85,B 0,C 180,E1 -1525.195,E2 -1525.195} C_VEL
LIN {X 0,Y 587.212,Z 552.899,A -85,B 0,C 180,E1 -1526.227,E2 -1526.227} C_VEL
LIN {X 0,Y 587.132,Z 555.811,A -85,B 0,C 180,E1 -1527.257,E2 -1527.257} C_VEL
LIN {X 0,Y 587.139,Z 557.202,A -85,B 0,C 180,E1 -1527.943,E2 -1527.943} C_VEL
LIN {X 0,Y 587.14,Z 558.785,A -85,B 0,C 180,E1 -1529.315,E2 -1529.315} C_VEL
LIN {X 0,Y 587.137,Z 559,A -85,B 0,C 180,E1 -1530.001,E2 -1530.001} C_VEL
LIN {X 0,Y 587.147,Z 558.184,A -85,B 0,C 180,E1 -1531.373,E2 -1531.373} C_VEL
LIN {X 0,Y 587.139,Z 557.199,A -85,B 0,C 180,E1 -1532.059,E2 -1532.059} C_VEL
LIN {X 0,Y 587.132,Z 555.807,A -85,B 0,C 180,E1 -1532.745,E2 -1532.745} C_VEL
LIN {X 0,Y 587.212,Z 552.893,A -85,B 0,C 180,E1 -1533.775,E2 -1533.775} C_VEL
LIN {X 0,Y 587.147,Z 548.945,A -85,B 0,C 180,E1 -1534.807,E2 -1534.807} C_VEL
LIN {X 0,Y 587.217,Z 542.872,A -85,B 0,C 180,E1 -1536.012,E2 -1536.012} C_VEL
LIN {X 0,Y 587.246,Z 536.23,A -85,B 0,C 180,E1 -1537.047,E2 -1537.047} C_VEL
LIN {X 0,Y 587.298,Z 527.982,A -85,B 0,C 180,E1 -1538.084,E2 -1538.084} C_VEL
LIN {X 0,Y 587.357,Z 517.591,A -85,B 0,C 180,E1 -1539.123,E2 -1539.123} C_VEL
LIN {X 0,Y 587.432,Z 507.916,A -85,B 0,C 180,E1 -1539.904,E2 -1539.904} C_VEL
LIN {X 0,Y 587.519,Z 497.312,A -85,B 0,C 180,E1 -1540.599,E2 -1540.599} C_VEL
LIN {X 0,Y 587.595,Z 485.31,A -85,B 0,C 180,E1 -1541.215,E2 -1541.215} C_VEL
LIN {X 0,Y 587.601,Z 473.213,A -85,B 0,C 180,E1 -1541.687,E2 -1541.687} C_VEL
LIN {X 0,Y 587.676,Z 460.483,A -85,B 0,C 180,E1 -1542.037,E2 -1542.037} C_VEL
LIN {X 0,Y 587.747,Z 447.236,A -85,B 0,C 180,E1 -1542.255,E2 -1542.255} C_VEL
LIN {X 0,Y 587.714,Z 348.861,A -85,B 0,C 180,E1 -1543.463,E2 -1543.463} C_VEL
LIN {X 0,Y 587.392,Z 346.606,A -85,B 0,C 180,E1 -1543.515,E2 -1543.515} C_VEL
LIN {X 0,Y 587.47,Z 328.646,A -85,B 0,C 180,E1 -1545.972,E2 -1545.972} C_VEL
LIN {X 0,Y 587.633,Z 309.229,A -85,B 0,C 180,E1 -1548.659,E2 -1548.659} C_VEL
LIN {X 0,Y 587.804,Z 288.493,A -85,B 0,C 180,E1 -1551.576,E2 -1551.576} C_VEL
LIN {X 0,Y 587.806,Z 279.777,A -85,B 0,C 180,E1 -1552.821,E2 -1552.821} C_VEL
LIN {X 0,Y 587.324,Z 277.326,A -85,B 0,C 180,E1 -1553.207,E2 -1553.207} C_VEL
LIN {X 0,Y 587.326,Z 277.323,A -85,B 0,C 180,E1 -1555.518,E2 -1555.518} C_VEL
LIN {X 0,Y 587.345,Z 277.323,A -85,B 0,C 180,E1 -1557.819,E2 -1557.819} C_VEL
LIN {X 0,Y 587.342,Z 277.321,A -85,B 0,C 180,E1 -1560.51,E2 -1560.51} C_VEL
LIN {X 0,Y 587.332,Z 277.318,A -85,B 0,C 180,E1 -1563.398,E2 -1563.398} C_VEL
LIN {X 0,Y 587.294,Z 277.326,A -85,B 0,C 180,E1 -1565.901,E2 -1565.901} C_VEL
LIN {X 0,Y 587.324,Z 277.329,A -85,B 0,C 180,E1 -1568.481,E2 -1568.481} C_VEL
LIN {X 0,Y 587.339,Z 277.318,A -85,B 0,C 180,E1 -1571.157,E2 -1571.157} C_VEL
LIN {X 0,Y 587.317,Z 277.322,A -85,B 0,C 180,E1 -1574.112,E2 -1574.112} C_VEL
LIN {X 0,Y 587.319,Z 277.325,A -85,B 0,C 180,E1 -1576.994,E2 -1576.994} C_VEL
LIN {X 0,Y 587.314,Z 277.32,A -85,B 0,C 180,E1 -1579.745,E2 -1579.745} C_VEL
LIN {X 0,Y 587.348,Z 277.319,A -85,B 0,C 180,E1 -1582.392,E2 -1582.392} C_VEL
LIN {X 0,Y 587.345,Z 277.317,A -85,B 0,C 180,E1 -1585.654,E2 -1585.654} C_VEL
LIN {X 0,Y 587.342,Z 277.316,A -85,B 0,C 180,E1 -1588.231,E2 -1588.231} C_VEL
LIN {X 0,Y 587.353,Z 277.321,A -85,B 0,C 180,E1 -1590.867,E2 -1590.867} C_VEL
LIN {X 0,Y 587.344,Z 277.318,A -85,B 0,C 180,E1 -1593.823,E2 -1593.823} C_VEL
LIN {X 0,Y 587.323,Z 277.32,A -85,B 0,C 180,E1 -1595.993,E2 -1595.993} C_VEL
LIN {X 0,Y 587.32,Z 277.319,A -85,B 0,C 180,E1 -1598.225,E2 -1598.225} C_VEL
LIN {X 0,Y 587.352,Z 277.32,A -85,B 0,C 180,E1 -1601.151,E2 -1601.151} C_VEL
LIN {X 0,Y 587.321,Z 277.322,A -85,B 0,C 180,E1 -1604.025,E2 -1604.025} C_VEL
LIN {X 0,Y 587.359,Z 277.317,A -85,B 0,C 180,E1 -1606.154,E2 -1606.154} C_VEL
LIN {X 0,Y 587.342,Z 277.317,A -85,B 0,C 180,E1 -1608.962,E2 -1608.962} C_VEL
LIN {X 0,Y 587.344,Z 277.326,A -85,B 0,C 180,E1 -1611.744,E2 -1611.744} C_VEL
LIN {X 0,Y 587.359,Z 277.316,A -85,B 0,C 180,E1 -1614.507,E2 -1614.507} C_VEL
LIN {X 0,Y 587.367,Z 277.314,A -85,B 0,C 180,E1 -1617.257,E2 -1617.257} C_VEL
LIN {X 0,Y 587.383,Z 277.32,A -85,B 0,C 180,E1 -1620,E2 -1620} C_VEL
LIN {X 0,Y 587.372,Z 277.315,A -85,B 0,C 180,E1 -1622.743,E2 -1622.743} C_VEL
LIN {X 0,Y 587.356,Z 277.315,A -85,B 0,C 180,E1 -1625.493,E2 -1625.493} C_VEL
LIN {X 0,Y 587.343,Z 277.325,A -85,B 0,C 180,E1 -1628.255,E2 -1628.255} C_VEL
LIN {X 0,Y 587.353,Z 277.316,A -85,B 0,C 180,E1 -1631.133,E2 -1631.133} C_VEL
LIN {X 0,Y 587.36,Z 277.319,A -85,B 0,C 180,E1 -1634.257,E2 -1634.257} C_VEL
LIN {X 0,Y 587.349,Z 277.316,A -85,B 0,C 180,E1 -1637.406,E2 -1637.406} C_VEL
LIN {X 0,Y 587.304,Z 277.324,A -85,B 0,C 180,E1 -1638.306,E2 -1638.306} C_VEL
LIN {X 0,Y 586.666,Z 277.409,A -85,B 0,C 180,E1 -1638.878,E2 -1638.878} C_VEL
LIN {X 0,Y 583.848,Z 277.761,A -85,B 0,C 180,E1 -1639.807,E2 -1639.807} C_VEL
LIN {X 0,Y 581.438,Z 278.06,A -85,B 0,C 180,E1 -1640.554,E2 -1640.554} C_VEL
LIN {X 0,Y 580.382,Z 278.189,A -85,B 0,C 180,E1 -1641.13,E2 -1641.13} C_VEL
LIN {X 0,Y 580.285,Z 278.198,A -85,B 0,C 180,E1 -1641.326,E2 -1641.326} C_VEL
LIN {X 0,Y 580.272,Z 278.198,A -85,B 0,C 180,E1 -1643.558,E2 -1643.558} C_VEL
LIN {X 0,Y 580.293,Z 278.194,A -85,B 0,C 180,E1 -1645.849,E2 -1645.849} C_VEL
LIN {X 0,Y 580.3,Z 278.194,A -85,B 0,C 180,E1 -1648.185,E2 -1648.185} C_VEL
LIN {X 0,Y 580.287,Z 278.199,A -85,B 0,C 180,E1 -1650.694,E2 -1650.694} C_VEL
LIN {X 0,Y 580.305,Z 278.202,A -85,B 0,C 180,E1 -1653.316,E2 -1653.316} C_VEL
LIN {X 0,Y 580.247,Z 278.203,A -85,B 0,C 180,E1 -1655.756,E2 -1655.756} C_VEL
LIN {X 0,Y 580.288,Z 278.195,A -85,B 0,C 180,E1 -1658.146,E2 -1658.146} C_VEL
LIN {X 0,Y 580.299,Z 278.195,A -85,B 0,C 180,E1 -1660.843,E2 -1660.843} C_VEL
LIN {X 0,Y 580.276,Z 278.205,A -85,B 0,C 180,E1 -1663.658,E2 -1663.658} C_VEL
LIN {X 0,Y 580.277,Z 278.196,A -85,B 0,C 180,E1 -1666.609,E2 -1666.609} C_VEL
LIN {X 0,Y 580.3,Z 278.196,A -85,B 0,C 180,E1 -1669.156,E2 -1669.156} C_VEL
LIN {X 0,Y 580.292,Z 278.204,A -85,B 0,C 180,E1 -1671.927,E2 -1671.927} C_VEL
LIN {X 0,Y 580.252,Z 278.202,A -85,B 0,C 180,E1 -1674.452,E2 -1674.452} C_VEL
LIN {X 0,Y 580.291,Z 278.194,A -85,B 0,C 180,E1 -1676.974,E2 -1676.974} C_VEL
LIN {X 0,Y 580.298,Z 278.195,A -85,B 0,C 180,E1 -1679.424,E2 -1679.424} C_VEL
LIN {X 0,Y 580.301,Z 278.205,A -85,B 0,C 180,E1 -1682.141,E2 -1682.141} C_VEL
LIN {X 0,Y 580.325,Z 278.19,A -85,B 0,C 180,E1 -1685.269,E2 -1685.269} C_VEL
LIN {X 0,Y 580.272,Z 278.201,A -85,B 0,C 180,E1 -1687.947,E2 -1687.947} C_VEL
LIN {X 0,Y 580.304,Z 278.196,A -85,B 0,C 180,E1 -1690.913,E2 -1690.913} C_VEL
LIN {X 0,Y 580.275,Z 278.197,A -85,B 0,C 180,E1 -1693.825,E2 -1693.825} C_VEL
LIN {X 0,Y 580.32,Z 278.193,A -85,B 0,C 180,E1 -1695.982,E2 -1695.982} C_VEL
LIN {X 0,Y 580.308,Z 278.201,A -85,B 0,C 180,E1 -1698.826,E2 -1698.826} C_VEL
LIN {X 0,Y 580.313,Z 278.193,A -85,B 0,C 180,E1 -1701.643,E2 -1701.643} C_VEL
LIN {X 0,Y 580.276,Z 278.198,A -85,B 0,C 180,E1 -1703.741,E2 -1703.741} C_VEL
LIN {X 0,Y 580.332,Z 278.311,A -85,B 0,C 180,E1 -1706.028,E2 -1706.028} C_VEL
LIN {X 0,Y 580.438,Z 284.916,A -85,B 0,C 180,E1 -1707.223,E2 -1707.223} C_VEL
LIN {X 0,Y 580.353,Z 300.484,A -85,B 0,C 180,E1 -1709.999,E2 -1709.999} C_VEL
LIN {X 0,Y 580.272,Z 308.351,A -85,B 0,C 180,E1 -1711.387,E2 -1711.387} C_VEL
LIN {X 0,Y 580.972,Z 312.848,A -85,B 0,C 180,E1 -1711.472,E2 -1711.472} C_VEL
LIN {X 0,Y 580.714,Z 414.987,A -85,B 0,C 180,E1 -1712.752,E2 -1712.752} C_VEL
LIN {X 0,Y 580.689,Z 428.039,A -85,B 0,C 180,E1 -1713.056,E2 -1713.056} C_VEL
LIN {X 0,Y 580.645,Z 441.156,A -85,B 0,C 180,E1 -1713.512,E2 -1713.512} C_VEL
LIN {X 0,Y 580.526,Z 453.07,A -85,B 0,C 180,E1 -1714.077,E2 -1714.077} C_VEL
LIN {X 0,Y 580.388,Z 464.466,A -85,B 0,C 180,E1 -1714.774,E2 -1714.774} C_VEL
LIN {X 0,Y 580.361,Z 474.722,A -85,B 0,C 180,E1 -1715.558,E2 -1715.558} C_VEL
LIN {X 0,Y 580.294,Z 483.414,A -85,B 0,C 180,E1 -1716.374,E2 -1716.374} C_VEL
LIN {X 0,Y 580.216,Z 491.694,A -85,B 0,C 180,E1 -1717.306,E2 -1717.306} C_VEL
LIN {X 0,Y 580.141,Z 499.236,A -85,B 0,C 180,E1 -1718.358,E2 -1718.358} C_VEL
LIN {X 0,Y 580.133,Z 505.307,A -85,B 0,C 180,E1 -1719.412,E2 -1719.412} C_VEL
LIN {X 0,Y 580.1,Z 510.13,A -85,B 0,C 180,E1 -1720.469,E2 -1720.469} C_VEL
LIN {X 0,Y 580.071,Z 513.832,A -85,B 0,C 180,E1 -1721.53,E2 -1721.53} C_VEL
LIN {X 0,Y 580.049,Z 516.503,A -85,B 0,C 180,E1 -1722.596,E2 -1722.596} C_VEL
LIN {X 0,Y 580.058,Z 517.751,A -85,B 0,C 180,E1 -1723.308,E2 -1723.308} C_VEL
LIN {X 0,Y 580.046,Z 518.706,A -85,B 0,C 180,E1 -1724.234,E2 -1724.234} C_VEL
LIN {X 0,Y 580.019,Z 518.913,A -85,B 0,C 180,E1 -1725.459,E2 -1725.459} C_VEL
LIN {X 0,Y 580.035,Z 518.469,A -85,B 0,C 180,E1 -1726.18,E2 -1726.18} C_VEL
LIN {X 0,Y 580.034,Z 517.557,A -85,B 0,C 180,E1 -1726.904,E2 -1726.904} C_VEL
LIN {X 0,Y 580.045,Z 516.218,A -85,B 0,C 180,E1 -1727.631,E2 -1727.631} C_VEL
LIN {X 0,Y 580.066,Z 513.337,A -85,B 0,C 180,E1 -1728.722,E2 -1728.722} C_VEL
LIN {X 0,Y 580.101,Z 509.283,A -85,B 0,C 180,E1 -1729.828,E2 -1729.828} C_VEL
LIN {X 0,Y 580.105,Z 504.439,A -85,B 0,C 180,E1 -1730.846,E2 -1730.846} C_VEL
LIN {X 0,Y 580.157,Z 498.36,A -85,B 0,C 180,E1 -1731.869,E2 -1731.869} C_VEL
LIN {X 0,Y 580.204,Z 491.536,A -85,B 0,C 180,E1 -1732.805,E2 -1732.805} C_VEL
LIN {X 0,Y 580.271,Z 483.122,A -85,B 0,C 180,E1 -1733.746,E2 -1733.746} C_VEL
LIN {X 0,Y 580.365,Z 474.266,A -85,B 0,C 180,E1 -1734.57,E2 -1734.57} C_VEL
LIN {X 0,Y 580.478,Z 463.826,A -85,B 0,C 180,E1 -1735.358,E2 -1735.358} C_VEL
LIN {X 0,Y 580.535,Z 453.351,A -85,B 0,C 180,E1 -1735.997,E2 -1735.997} C_VEL
LIN {X 0,Y 580.666,Z 442.316,A -85,B 0,C 180,E1 -1736.529,E2 -1736.529} C_VEL
LIN {X 0,Y 580.704,Z 429.578,A -85,B 0,C 180,E1 -1736.989,E2 -1736.989} C_VEL
LIN {X 0,Y 580.773,Z 416.765,A -85,B 0,C 180,E1 -1737.302,E2 -1737.302} C_VEL
LIN {X 0,Y 580.863,Z 389.888,A -85,B 0,C 180,E1 -1737.663,E2 -1737.663} C_VEL
LIN {X 0,Y 580.859,Z 312.115,A -85,B 0,C 180,E1 -1738.63,E2 -1738.63} C_VEL
LIN {X 0,Y 580.297,Z 308.353,A -85,B 0,C 180,E1 -1738.702,E2 -1738.702} C_VEL
LIN {X 0,Y 580.386,Z 291.39,A -85,B 0,C 180,E1 -1741.708,E2 -1741.708} C_VEL
LIN {X 0,Y 580.424,Z 279.489,A -85,B 0,C 180,E1 -1743.846,E2 -1743.846} C_VEL
LIN {X 0,Y 580.24,Z 278.206,A -85,B 0,C 180,E1 -1744.12,E2 -1744.12} C_VEL
LIN {X 0,Y 580.267,Z 278.209,A -85,B 0,C 180,E1 -1747.269,E2 -1747.269} C_VEL
LIN {X 0,Y 580.259,Z 278.2,A -85,B 0,C 180,E1 -1750.267,E2 -1750.267} C_VEL
LIN {X 0,Y 580.231,Z 278.204,A -85,B 0,C 180,E1 -1752.709,E2 -1752.709} C_VEL
LIN {X 0,Y 580.233,Z 278.209,A -85,B 0,C 180,E1 -1755.611,E2 -1755.611} C_VEL
LIN {X 0,Y 580.236,Z 278.203,A -85,B 0,C 180,E1 -1758.227,E2 -1758.227} C_VEL
LIN {X 0,Y 580.247,Z 278.203,A -85,B 0,C 180,E1 -1760.963,E2 -1760.963} C_VEL
LIN {X 0,Y 580.226,Z 278.213,A -85,B 0,C 180,E1 -1763.593,E2 -1763.593} C_VEL
LIN {X 0,Y 580.291,Z 278.198,A -85,B 0,C 180,E1 -1766.144,E2 -1766.144} C_VEL
LIN {X 0,Y 580.256,Z 278.199,A -85,B 0,C 180,E1 -1768.613,E2 -1768.613} C_VEL
LIN {X 0,Y 580.27,Z 278.198,A -85,B 0,C 180,E1 -1771.023,E2 -1771.023} C_VEL
LIN {X 0,Y 580.247,Z 278.206,A -85,B 0,C 180,E1 -1774.149,E2 -1774.149} C_VEL
LIN {X 0,Y 580.259,Z 278.202,A -85,B 0,C 180,E1 -1776.441,E2 -1776.441} C_VEL
LIN {X 0,Y 580.251,Z 278.201,A -85,B 0,C 180,E1 -1779.436,E2 -1779.436} C_VEL
LIN {X 0,Y 580.25,Z 278.204,A -85,B 0,C 180,E1 -1781.645,E2 -1781.645} C_VEL
LIN {X 0,Y 580.239,Z 278.206,A -85,B 0,C 180,E1 -1783.825,E2 -1783.825} C_VEL
LIN {X 0,Y 580.301,Z 278.201,A -85,B 0,C 180,E1 -1785.983,E2 -1785.983} C_VEL
LIN {X 0,Y 580.289,Z 278.197,A -85,B 0,C 180,E1 -1788.827,E2 -1788.827} C_VEL
LIN {X 0,Y 580.309,Z 278.194,A -85,B 0,C 180,E1 -1791.644,E2 -1791.644} C_VEL
LIN {X 0,Y 580.314,Z 278.202,A -85,B 0,C 180,E1 -1794.44,E2 -1794.44} C_VEL
LIN {X 0,Y 580.319,Z 278.191,A -85,B 0,C 180,E1 -1797.224,E2 -1797.224} C_VEL
LIN {X 0,Y 580.324,Z 278.193,A -85,B 0,C 180,E1 -1800,E2 -1800} C_VEL
LIN {X 0,Y 580.34,Z 278.194,A -85,B 0,C 180,E1 -1802.777,E2 -1802.777} C_VEL
LIN {X 0,Y 580.31,Z 278.192,A -85,B 0,C 180,E1 -1805.56,E2 -1805.56} C_VEL
LIN {X 0,Y 580.318,Z 278.196,A -85,B 0,C 180,E1 -1808.356,E2 -1808.356} C_VEL
LIN {X 0,Y 580.32,Z 278.195,A -85,B 0,C 180,E1 -1811.209,E2 -1811.209} C_VEL
LIN {X 0,Y 580.301,Z 278.195,A -85,B 0,C 180,E1 -1814.339,E2 -1814.339} C_VEL
LIN {X 0,Y 580.298,Z 278.205,A -85,B 0,C 180,E1 -1816.914,E2 -1816.914} C_VEL
LIN {X 0,Y 580.292,Z 278.195,A -85,B 0,C 180,E1 -1819.823,E2 -1819.823} C_VEL
LIN {X 0,Y 580.284,Z 278.202,A -85,B 0,C 180,E1 -1822.803,E2 -1822.803} C_VEL
LIN {X 0,Y 580.298,Z 278.204,A -85,B 0,C 180,E1 -1825.08,E2 -1825.08} C_VEL
LIN {X 0,Y 580.286,Z 278.195,A -85,B 0,C 180,E1 -1827.86,E2 -1827.86} C_VEL
LIN {X 0,Y 580.288,Z 278.198,A -85,B 0,C 180,E1 -1830.698,E2 -1830.698} C_VEL
LIN {X 0,Y 580.295,Z 278.206,A -85,B 0,C 180,E1 -1833.318,E2 -1833.318} C_VEL
LIN {X 0,Y 580.315,Z 278.196,A -85,B 0,C 180,E1 -1835.768,E2 -1835.768} C_VEL
LIN {X 0,Y 580.28,Z 278.197,A -85,B 0,C 180,E1 -1838.147,E2 -1838.147} C_VEL
LIN {X 0,Y 580.292,Z 278.197,A -85,B 0,C 180,E1 -1840.844,E2 -1840.844} C_VEL
LIN {X 0,Y 580.279,Z 278.205,A -85,B 0,C 180,E1 -1843.658,E2 -1843.658} C_VEL
LIN {X 0,Y 580.278,Z 278.196,A -85,B 0,C 180,E1 -1846.61,E2 -1846.61} C_VEL
LIN {X 0,Y 580.295,Z 278.197,A -85,B 0,C 180,E1 -1849.158,E2 -1849.158} C_VEL
LIN {X 0,Y 580.285,Z 278.204,A -85,B 0,C 180,E1 -1851.928,E2 -1851.928} C_VEL
LIN {X 0,Y 580.28,Z 278.198,A -85,B 0,C 180,E1 -1854.456,E2 -1854.456} C_VEL
LIN {X 0,Y 580.286,Z 278.196,A -85,B 0,C 180,E1 -1856.977,E2 -1856.977} C_VEL
LIN {X 0,Y 580.295,Z 278.198,A -85,B 0,C 180,E1 -1859.427,E2 -1859.427} C_VEL
LIN {X 0,Y 580.317,Z 278.201,A -85,B 0,C 180,E1 -1862.138,E2 -1862.138} C_VEL
LIN {X 0,Y 580.319,Z 278.194,A -85,B 0,C 180,E1 -1865.271,E2 -1865.271} C_VEL
LIN {X 0,Y 580.308,Z 278.265,A -85,B 0,C 180,E1 -1866.66,E2 -1866.66} C_VEL
LIN {X 0,Y 580.969,Z 283.355,A -85,B 0,C 180,E1 -1867.415,E2 -1867.415} C_VEL
LIN {X 0,Y 580.753,Z 305.066,A -85,B 0,C 180,E1 -1870.521,E2 -1870.521} C_VEL
LIN {X 0,Y 580.544,Z 326.072,A -85,B 0,C 180,E1 -1873.473,E2 -1873.473} C_VEL
LIN {X 0,Y 580.398,Z 346.622,A -85,B 0,C 180,E1 -1876.321,E2 -1876.321} C_VEL
LIN {X 0,Y 580.987,Z 352.607,A -85,B 0,C 180,E1 -1876.424,E2 -1876.424} C_VEL
LIN {X 0,Y 580.785,Z 455.009,A -85,B 0,C 180,E1 -1877.709,E2 -1877.709} C_VEL
LIN {X 0,Y 580.729,Z 468.261,A -85,B 0,C 180,E1 -1878.018,E2 -1878.018} C_VEL
LIN {X 0,Y 580.652,Z 481.174,A -85,B 0,C 180,E1 -1878.468,E2 -1878.468} C_VEL
LIN {X 0,Y 580.551,Z 492.65,A -85,B 0,C 180,E1 -1879.01,E2 -1879.01} C_VEL
LIN {X 0,Y 580.42,Z 504.22,A -85,B 0,C 180,E1 -1879.713,E2 -1879.713} C_VEL
LIN {X 0,Y 580.342,Z 514.614,A -85,B 0,C 180,E1 -1880.504,E2 -1880.504} C_VEL
LIN {X 0,Y 580.262,Z 523.067,A -85,B 0,C 180,E1 -1881.293,E2 -1881.293} C_VEL
LIN {X 0,Y 580.221,Z 530.97,A -85,B 0,C 180,E1 -1882.169,E2 -1882.169} C_VEL
LIN {X 0,Y 580.155,Z 538.642,A -85,B 0,C 180,E1 -1883.22,E2 -1883.22} C_VEL
LIN {X 0,Y 580.139,Z 545.686,A -85,B 0,C 180,E1 -1884.44,E2 -1884.44} C_VEL
LIN {X 0,Y 580.108,Z 550.376,A -85,B 0,C 180,E1 -1885.485,E2 -1885.485} C_VEL
LIN {X 0,Y 580.122,Z 553.96,A -85,B 0,C 180,E1 -1886.528,E2 -1886.528} C_VEL
LIN {X 0,Y 580.043,Z 555.811,A -85,B 0,C 180,E1 -1887.223,E2 -1887.223} C_VEL
LIN {X 0,Y 580.038,Z 557.201,A -85,B 0,C 180,E1 -1887.918,E2 -1887.918} C_VEL
LIN {X 0,Y 580.04,Z 558.785,A -85,B 0,C 180,E1 -1889.307,E2 -1889.307} C_VEL
LIN {X 0,Y 580.037,Z 559,A -85,B 0,C 180,E1 -1890.001,E2 -1890.001} C_VEL
LIN {X 0,Y 580.046,Z 558.185,A -85,B 0,C 180,E1 -1891.39,E2 -1891.39} C_VEL
LIN {X 0,Y 580.038,Z 557.198,A -85,B 0,C 180,E1 -1892.084,E2 -1892.084} C_VEL
LIN {X 0,Y 580.043,Z 555.807,A -85,B 0,C 180,E1 -1892.779,E2 -1892.779} C_VEL
LIN {X 0,Y 580.109,Z 552.893,A -85,B 0,C 180,E1 -1893.822,E2 -1893.822} C_VEL
LIN {X 0,Y 580.053,Z 548.945,A -85,B 0,C 180,E1 -1894.866,E2 -1894.866} C_VEL
LIN {X 0,Y 580.14,Z 542.871,A -85,B 0,C 180,E1 -1896.086,E2 -1896.086} C_VEL
LIN {X 0,Y 580.185,Z 536.231,A -85,B 0,C 180,E1 -1897.133,E2 -1897.133} C_VEL
LIN {X 0,Y 580.247,Z 527.982,A -85,B 0,C 180,E1 -1898.183,E2 -1898.183} C_VEL
LIN {X 0,Y 580.333,Z 517.591,A -85,B 0,C 180,E1 -1899.235,E2 -1899.235} C_VEL
LIN {X 0,Y 580.437,Z 507.914,A -85,B 0,C 180,E1 -1900.025,E2 -1900.025} C_VEL
LIN {X 0,Y 580.531,Z 497.311,A -85,B 0,C 180,E1 -1900.728,E2 -1900.728} C_VEL
LIN {X 0,Y 580.614,Z 485.476,A -85,B 0,C 180,E1 -1901.344,E2 -1901.344} C_VEL
LIN {X 0,Y 580.671,Z 473.146,A -85,B 0,C 180,E1 -1901.83,E2 -1901.83} C_VEL
LIN {X 0,Y 580.756,Z 460.482,A -85,B 0,C 180,E1 -1902.183,E2 -1902.183} C_VEL
LIN {X 0,Y 580.836,Z 447.236,A -85,B 0,C 180,E1 -1902.403,E2 -1902.403} C_VEL
LIN {X 0,Y 580.799,Z 349.53,A -85,B 0,C 180,E1 -1903.619,E2 -1903.619} C_VEL
LIN {X 0,Y 580.398,Z 346.606,A -85,B 0,C 180,E1 -1903.681,E2 -1903.681} C_VEL
LIN {X 0,Y 580.546,Z 326.057,A -85,B 0,C 180,E1 -1906.529,E2 -1906.529} C_VEL
LIN {X 0,Y 580.756,Z 305.059,A -85,B 0,C 180,E1 -1909.48,E2 -1909.48} C_VEL
LIN {X 0,Y 580.962,Z 284.634,A -85,B 0,C 180,E1 -1912.4,E2 -1912.4} C_VEL
LIN {X 0,Y 580.635,Z 279.96,A -85,B 0,C 180,E1 -1913.087,E2 -1913.087} C_VEL
LIN {X 0,Y 580.277,Z 278.205,A -85,B 0,C 180,E1 -1913.379,E2 -1913.379} C_VEL
LIN {X 0,Y 580.28,Z 278.206,A -85,B 0,C 180,E1 -1915.85,E2 -1915.85} C_VEL
LIN {X 0,Y 580.299,Z 278.203,A -85,B 0,C 180,E1 -1918.186,E2 -1918.186} C_VEL
LIN {X 0,Y 580.289,Z 278.197,A -85,B 0,C 180,E1 -1920.695,E2 -1920.695} C_VEL
LIN {X 0,Y 580.288,Z 278.195,A -85,B 0,C 180,E1 -1923.314,E2 -1923.314} C_VEL
LIN {X 0,Y 580.248,Z 278.202,A -85,B 0,C 180,E1 -1925.756,E2 -1925.756} C_VEL
LIN {X 0,Y 580.289,Z 278.201,A -85,B 0,C 180,E1 -1928.147,E2 -1928.147} C_VEL
LIN {X 0,Y 580.301,Z 278.198,A -85,B 0,C 180,E1 -1930.844,E2 -1930.844} C_VEL
LIN {X 0,Y 580.277,Z 278.196,A -85,B 0,C 180,E1 -1933.659,E2 -1933.659} C_VEL
LIN {X 0,Y 580.28,Z 278.206,A -85,B 0,C 180,E1 -1936.61,E2 -1936.61} C_VEL
LIN {X 0,Y 580.301,Z 278.198,A -85,B 0,C 180,E1 -1939.157,E2 -1939.157} C_VEL
LIN {X 0,Y 580.293,Z 278.194,A -85,B 0,C 180,E1 -1941.928,E2 -1941.928} C_VEL
LIN {X 0,Y 580.254,Z 278.202,A -85,B 0,C 180,E1 -1944.453,E2 -1944.453} C_VEL
LIN {X 0,Y 580.293,Z 278.205,A -85,B 0,C 180,E1 -1946.975,E2 -1946.975} C_VEL
LIN {X 0,Y 580.3,Z 278.199,A -85,B 0,C 180,E1 -1949.425,E2 -1949.425} C_VEL
LIN {X 0,Y 580.296,Z 278.194,A -85,B 0,C 180,E1 -1952.143,E2 -1952.143} C_VEL
LIN {X 0,Y 580.307,Z 278.197,A -85,B 0,C 180,E1 -1954.92,E2 -1954.92} C_VEL
LIN {X 0,Y 580.272,Z 278.199,A -85,B 0,C 180,E1 -1957.947,E2 -1957.947} C_VEL
LIN {X 0,Y 580.302,Z 278.195,A -85,B 0,C 180,E1 -1960.913,E2 -1960.913} C_VEL
LIN {X 0,Y 580.272,Z 278.203,A -85,B 0,C 180,E1 -1963.825,E2 -1963.825} C_VEL
LIN {X 0,Y 580.328,Z 278.195,A -85,B 0,C 180,E1 -1965.983,E2 -1965.983} C_VEL
LIN {X 0,Y 580.31,Z 278.192,A -85,B 0,C 180,E1 -1968.827,E2 -1968.827} C_VEL
LIN {X 0,Y 580.313,Z 278.199,A -85,B 0,C 180,E1 -1971.644,E2 -1971.644} C_VEL
LIN {X 0,Y 580.324,Z 278.193,A -85,B 0,C 180,E1 -1974.44,E2 -1974.44} C_VEL
LIN {X 0,Y 580.335,Z 278.189,A -85,B 0,C 180,E1 -1977.223,E2 -1977.223} C_VEL
LIN {X 0,Y 580.353,Z 278.196,A -85,B 0,C 180,E1 -1980,E2 -1980} C_VEL
LIN {X 0,Y 580.339,Z 278.191,A -85,B 0,C 180,E1 -1982.776,E2 -1982.776} C_VEL
LIN {X 0,Y 580.322,Z 278.191,A -85,B 0,C 180,E1 -1985.56,E2 -1985.56} C_VEL
LIN {X 0,Y 580.326,Z 278.191,A -85,B 0,C 180,E1 -1987.655,E2 -1987.655} C_VEL
LIN {X 0,Y 580.3,Z 278.205,A -85,B 0,C 180,E1 -1990.467,E2 -1990.467} C_VEL
LIN {X 0,Y 580.304,Z 278.203,A -85,B 0,C 180,E1 -1992.591,E2 -1992.591} C_VEL
LIN {X 0,Y 580.289,Z 278.203,A -85,B 0,C 180,E1 -1994.734,E2 -1994.734} C_VEL
LIN {X 0,Y 580.291,Z 278.194,A -85,B 0,C 180,E1 -1997.624,E2 -1997.624} C_VEL
LIN {X 0,Y 580.288,Z 278.195,A -85,B 0,C 180,E1 -1999.823,E2 -1999.823} C_VEL
LIN {X 0,Y 580.285,Z 278.198,A -85,B 0,C 180,E1 -2001.326,E2 -2001.326} C_VEL
LIN {X 0,Y 579.584,Z 278.285,A -85,B 0,C 180,E1 -2001.905,E2 -2001.905} C_VEL
LIN {X 0,Y 576.704,Z 278.653,A -85,B 0,C 180,E1 -2002.845,E2 -2002.845} C_VEL
LIN {X 0,Y 574.31,Z 278.944,A -85,B 0,C 180,E1 -2003.601,E2 -2003.601} C_VEL
LIN {X 0,Y 573.315,Z 279.065,A -85,B 0,C 180,E1 -2004.185,E2 -2004.185} C_VEL
LIN {X 0,Y 573.25,Z 279.074,A -85,B 0,C 180,E1 -2004.382,E2 -2004.382} C_VEL
LIN {X 0,Y 573.254,Z 279.082,A -85,B 0,C 180,E1 -2006.976,E2 -2006.976} C_VEL
LIN {X 0,Y 573.249,Z 279.076,A -85,B 0,C 180,E1 -2009.488,E2 -2009.488} C_VEL
LIN {X 0,Y 573.255,Z 279.073,A -85,B 0,C 180,E1 -2012.645,E2 -2012.645} C_VEL
LIN {X 0,Y 573.208,Z 279.087,A -85,B 0,C 180,E1 -2015.188,E2 -2015.188} C_VEL
LIN {X 0,Y 573.234,Z 279.077,A -85,B 0,C 180,E1 -2017.808,E2 -2017.808} C_VEL
LIN {X 0,Y 573.248,Z 279.072,A -85,B 0,C 180,E1 -2020.525,E2 -2020.525} C_VEL
LIN {X 0,Y 573.24,Z 279.081,A -85,B 0,C 180,E1 -2023.359,E2 -2023.359} C_VEL
LIN {X 0,Y 573.24,Z 279.073,A -85,B 0,C 180,E1 -2026.64,E2 -2026.64} C_VEL
LIN {X 0,Y 573.248,Z 279.078,A -85,B 0,C 180,E1 -2029.474,E2 -2029.474} C_VEL
LIN {X 0,Y 573.238,Z 279.078,A -85,B 0,C 180,E1 -2032.192,E2 -2032.192} C_VEL
LIN {X 0,Y 573.237,Z 279.074,A -85,B 0,C 180,E1 -2035.228,E2 -2035.228} C_VEL
LIN {X 0,Y 573.251,Z 279.078,A -85,B 0,C 180,E1 -2037.772,E2 -2037.772} C_VEL
LIN {X 0,Y 573.267,Z 279.072,A -85,B 0,C 180,E1 -2040.633,E2 -2040.633} C_VEL
LIN {X 0,Y 573.254,Z 279.071,A -85,B 0,C 180,E1 -2043.023,E2 -2043.023} C_VEL
LIN {X 0,Y 573.277,Z 279.068,A -85,B 0,C 180,E1 -2045.365,E2 -2045.365} C_VEL
LIN {X 0,Y 573.231,Z 279.084,A -85,B 0,C 180,E1 -2048.419,E2 -2048.419} C_VEL
LIN {X 0,Y 573.282,Z 279.073,A -85,B 0,C 180,E1 -2050.727,E2 -2050.727} C_VEL
LIN {X 0,Y 573.249,Z 279.072,A -85,B 0,C 180,E1 -2053.621,E2 -2053.621} C_VEL
LIN {X 0,Y 573.268,Z 279.07,A -85,B 0,C 180,E1 -2055.806,E2 -2055.806} C_VEL
LIN {X 0,Y 573.266,Z 279.08,A -85,B 0,C 180,E1 -2058.744,E2 -2058.744} C_VEL
LIN {X 0,Y 573.257,Z 279.072,A -85,B 0,C 180,E1 -2061.539,E2 -2061.539} C_VEL
LIN {X 0,Y 573.239,Z 279.075,A -85,B 0,C 180,E1 -2063.664,E2 -2063.664} C_VEL
LIN {X 0,Y 573.29,Z 279.248,A -85,B 0,C 180,E1 -2065.957,E2 -2065.957} C_VEL
LIN {X 0,Y 573.435,Z 284.036,A -85,B 0,C 180,E1 -2066.837,E2 -2066.837} C_VEL
LIN {X 0,Y 573.331,Z 297.628,A -85,B 0,C 180,E1 -2069.297,E2 -2069.297} C_VEL
LIN {X 0,Y 573.231,Z 308.421,A -85,B 0,C 180,E1 -2071.228,E2 -2071.228} C_VEL
LIN {X 0,Y 574.087,Z 313.498,A -85,B 0,C 180,E1 -2071.314,E2 -2071.314} C_VEL
LIN {X 0,Y 573.775,Z 415.429,A -85,B 0,C 180,E1 -2072.61,E2 -2072.61} C_VEL
LIN {X 0,Y 573.736,Z 429.083,A -85,B 0,C 180,E1 -2072.939,E2 -2072.939} C_VEL
LIN {X 0,Y 573.689,Z 441.372,A -85,B 0,C 180,E1 -2073.379,E2 -2073.379} C_VEL
LIN {X 0,Y 573.533,Z 453.232,A -85,B 0,C 180,E1 -2073.951,E2 -2073.951} C_VEL
LIN {X 0,Y 573.376,Z 464.601,A -85,B 0,C 180,E1 -2074.657,E2 -2074.657} C_VEL
LIN {X 0,Y 573.331,Z 474.836,A -85,B 0,C 180,E1 -2075.45,E2 -2075.45} C_VEL
LIN {X 0,Y 573.241,Z 484.069,A -85,B 0,C 180,E1 -2076.334,E2 -2076.334} C_VEL
LIN {X 0,Y 573.147,Z 491.768,A -85,B 0,C 180,E1 -2077.219,E2 -2077.219} C_VEL
LIN {X 0,Y 573.092,Z 499.29,A -85,B 0,C 180,E1 -2078.284,E2 -2078.284} C_VEL
LIN {X 0,Y 573.031,Z 506.265,A -85,B 0,C 180,E1 -2079.529,E2 -2079.529} C_VEL
LIN {X 0,Y 573.027,Z 510.878,A -85,B 0,C 180,E1 -2080.6,E2 -2080.6} C_VEL
LIN {X 0,Y 572.987,Z 514.395,A -85,B 0,C 180,E1 -2081.675,E2 -2081.675} C_VEL
LIN {X 0,Y 572.945,Z 516.889,A -85,B 0,C 180,E1 -2082.755,E2 -2082.755} C_VEL
LIN {X 0,Y 572.967,Z 518,A -85,B 0,C 180,E1 -2083.476,E2 -2083.476} C_VEL
LIN {X 0,Y 572.958,Z 518.756,A -85,B 0,C 180,E1 -2084.298,E2 -2084.298} C_VEL
LIN {X 0,Y 572.915,Z 518.846,A -85,B 0,C 180,E1 -2085.656,E2 -2085.656} C_VEL
LIN {X 0,Y 572.935,Z 517.595,A -85,B 0,C 180,E1 -2086.903,E2 -2086.903} C_VEL
LIN {X 0,Y 572.953,Z 515.81,A -85,B 0,C 180,E1 -2087.857,E2 -2087.857} C_VEL
LIN {X 0,Y 572.967,Z 511.971,A -85,B 0,C 180,E1 -2089.182,E2 -2089.182} C_VEL
LIN {X 0,Y 573.011,Z 506.745,A -85,B 0,C 180,E1 -2090.459,E2 -2090.459} C_VEL
LIN {X 0,Y 573.087,Z 500.687,A -85,B 0,C 180,E1 -2091.585,E2 -2091.585} C_VEL
LIN {X 0,Y 573.133,Z 492.917,A -85,B 0,C 180,E1 -2092.721,E2 -2092.721} C_VEL
LIN {X 0,Y 573.225,Z 484.874,A -85,B 0,C 180,E1 -2093.672,E2 -2093.672} C_VEL
LIN {X 0,Y 573.332,Z 474.954,A -85,B 0,C 180,E1 -2094.63,E2 -2094.63} C_VEL
LIN {X 0,Y 573.458,Z 463.67,A -85,B 0,C 180,E1 -2095.496,E2 -2095.496} C_VEL
LIN {X 0,Y 573.554,Z 452.598,A -85,B 0,C 180,E1 -2096.174,E2 -2096.174} C_VEL
LIN {X 0,Y 573.699,Z 440.091,A -85,B 0,C 180,E1 -2096.762,E2 -2096.762} C_VEL
LIN {X 0,Y 573.781,Z 426.762,A -85,B 0,C 180,E1 -2097.218,E2 -2097.218} C_VEL
LIN {X 0,Y 573.857,Z 413.594,A -85,B 0,C 180,E1 -2097.511,E2 -2097.511} C_VEL
LIN {X 0,Y 573.916,Z 312.533,A -85,B 0,C 180,E1 -2098.792,E2 -2098.792} C_VEL
LIN {X 0,Y 573.254,Z 308.343,A -85,B 0,C 180,E1 -2098.875,E2 -2098.875} C_VEL
LIN {X 0,Y 573.375,Z 292.013,A -85,B 0,C 180,E1 -2101.805,E2 -2101.805} C_VEL
LIN {X 0,Y 573.411,Z 280.483,A -85,B 0,C 180,E1 -2103.903,E2 -2103.903} C_VEL
LIN {X 0,Y 573.192,Z 279.084,A -85,B 0,C 180,E1 -2104.176,E2 -2104.176} C_VEL
LIN {X 0,Y 573.218,Z 279.087,A -85,B 0,C 180,E1 -2107.161,E2 -2107.161} C_VEL
LIN {X 0,Y 573.208,Z 279.083,A -85,B 0,C 180,E1 -2109.608,E2 -2109.608} C_VEL
LIN {X 0,Y 573.196,Z 279.08,A -85,B 0,C 180,E1 -2112.637,E2 -2112.637} C_VEL
LIN {X 0,Y 573.2,Z 279.084,A -85,B 0,C 180,E1 -2115.663,E2 -2115.663} C_VEL
LIN {X 0,Y 573.187,Z 279.08,A -85,B 0,C 180,E1 -2118.41,E2 -2118.41} C_VEL
LIN {X 0,Y 573.219,Z 279.076,A -85,B 0,C 180,E1 -2120.569,E2 -2120.569} C_VEL
LIN {X 0,Y 573.204,Z 279.081,A -85,B 0,C 180,E1 -2123.074,E2 -2123.074} C_VEL
LIN {X 0,Y 573.243,Z 279.082,A -85,B 0,C 180,E1 -2125.67,E2 -2125.67} C_VEL
LIN {X 0,Y 573.223,Z 279.078,A -85,B 0,C 180,E1 -2128.184,E2 -2128.184} C_VEL
LIN {X 0,Y 573.243,Z 279.073,A -85,B 0,C 180,E1 -2130.633,E2 -2130.633} C_VEL
LIN {X 0,Y 573.191,Z 279.084,A -85,B 0,C 180,E1 -2133.513,E2 -2133.513} C_VEL
LIN {X 0,Y 573.214,Z 279.084,A -85,B 0,C 180,E1 -2136.134,E2 -2136.134} C_VEL
LIN {X 0,Y 573.231,Z 279.074,A -85,B 0,C 180,E1 -2139.173,E2 -2139.173} C_VEL
LIN {X 0,Y 573.201,Z 279.08,A -85,B 0,C 180,E1 -2141.411,E2 -2141.411} C_VEL
LIN {X 0,Y 573.212,Z 279.079,A -85,B 0,C 180,E1 -2143.621,E2 -2143.621} C_VEL
LIN {X 0,Y 573.243,Z 279.078,A -85,B 0,C 180,E1 -2145.806,E2 -2145.806} C_VEL
LIN {X 0,Y 573.247,Z 279.075,A -85,B 0,C 180,E1 -2148.745,E2 -2148.745} C_VEL
LIN {X 0,Y 573.266,Z 279.071,A -85,B 0,C 180,E1 -2151.54,E2 -2151.54} C_VEL
LIN {X 0,Y 573.278,Z 279.079,A -85,B 0,C 180,E1 -2154.372,E2 -2154.372} C_VEL
LIN {X 0,Y 573.287,Z 279.067,A -85,B 0,C 180,E1 -2157.189,E2 -2157.189} C_VEL
LIN {X 0,Y 573.295,Z 279.069,A -85,B 0,C 180,E1 -2160,E2 -2160} C_VEL
LIN {X 0,Y 573.304,Z 279.07,A -85,B 0,C 180,E1 -2162.811,E2 -2162.811} C_VEL
LIN {X 0,Y 573.276,Z 279.069,A -85,B 0,C 180,E1 -2165.628,E2 -2165.628} C_VEL
LIN {X 0,Y 573.276,Z 279.074,A -85,B 0,C 180,E1 -2168.46,E2 -2168.46} C_VEL
LIN {X 0,Y 573.285,Z 279.07,A -85,B 0,C 180,E1 -2171.312,E2 -2171.312} C_VEL
LIN {X 0,Y 573.267,Z 279.072,A -85,B 0,C 180,E1 -2174.425,E2 -2174.425} C_VEL
LIN {X 0,Y 573.244,Z 279.079,A -85,B 0,C 180,E1 -2177.112,E2 -2177.112} C_VEL
LIN {X 0,Y 573.239,Z 279.073,A -85,B 0,C 180,E1 -2180.077,E2 -2180.077} C_VEL
LIN {X 0,Y 573.221,Z 279.085,A -85,B 0,C 180,E1 -2183.1,E2 -2183.1} C_VEL
LIN {X 0,Y 573.246,Z 279.078,A -85,B 0,C 180,E1 -2185.411,E2 -2185.411} C_VEL
LIN {X 0,Y 573.241,Z 279.072,A -85,B 0,C 180,E1 -2188.03,E2 -2188.03} C_VEL
LIN {X 0,Y 573.233,Z 279.079,A -85,B 0,C 180,E1 -2190.886,E2 -2190.886} C_VEL
LIN {X 0,Y 573.278,Z 279.076,A -85,B 0,C 180,E1 -2193.529,E2 -2193.529} C_VEL
LIN {X 0,Y 573.25,Z 279.073,A -85,B 0,C 180,E1 -2196.049,E2 -2196.049} C_VEL
LIN {X 0,Y 573.24,Z 279.074,A -85,B 0,C 180,E1 -2198.702,E2 -2198.702} C_VEL
LIN {X 0,Y 573.246,Z 279.082,A -85,B 0,C 180,E1 -2201.597,E2 -2201.597} C_VEL
LIN {X 0,Y 573.231,Z 279.075,A -85,B 0,C 180,E1 -2204.334,E2 -2204.334} C_VEL
LIN {X 0,Y 573.237,Z 279.079,A -85,B 0,C 180,E1 -2207.359,E2 -2207.359} C_VEL
LIN {X 0,Y 573.241,Z 279.074,A -85,B 0,C 180,E1 -2210.394,E2 -2210.394} C_VEL
LIN {X 0,Y 573.251,Z 279.073,A -85,B 0,C 180,E1 -2213.079,E2 -2213.079} C_VEL
LIN {X 0,Y 573.263,Z 279.079,A -85,B 0,C 180,E1 -2215.673,E2 -2215.673} C_VEL
LIN {X 0,Y 573.237,Z 279.08,A -85,B 0,C 180,E1 -2218.186,E2 -2218.186} C_VEL
LIN {X 0,Y 573.261,Z 279.073,A -85,B 0,C 180,E1 -2220.636,E2 -2220.636} C_VEL
LIN {X 0,Y 573.248,Z 279.074,A -85,B 0,C 180,E1 -2223.025,E2 -2223.025} C_VEL
LIN {X 0,Y 573.273,Z 279.073,A -85,B 0,C 180,E1 -2225.367,E2 -2225.367} C_VEL
LIN {X 0,Y 573.255,Z 279.142,A -85,B 0,C 180,E1 -2226.527,E2 -2226.527} C_VEL
LIN {X 0,Y 574.017,Z 284.43,A -85,B 0,C 180,E1 -2227.316,E2 -2227.316} C_VEL
LIN {X 0,Y 573.815,Z 304.068,A -85,B 0,C 180,E1 -2230.132,E2 -2230.132} C_VEL
LIN {X 0,Y 573.586,Z 324.249,A -85,B 0,C 180,E1 -2233.008,E2 -2233.008} C_VEL
LIN {X 0,Y 573.416,Z 346.46,A -85,B 0,C 180,E1 -2236.129,E2 -2236.129} C_VEL
LIN {X 0,Y 573.601,Z 348.135,A -85,B 0,C 180,E1 -2236.19,E2 -2236.19} C_VEL
LIN {X 0,Y 574.083,Z 352.607,A -85,B 0,C 180,E1 -2236.258,E2 -2236.258} C_VEL
LIN {X 0,Y 573.865,Z 455.009,A -85,B 0,C 180,E1 -2237.558,E2 -2237.558} C_VEL
LIN {X 0,Y 573.787,Z 468.26,A -85,B 0,C 180,E1 -2237.871,E2 -2237.871} C_VEL
LIN {X 0,Y 573.685,Z 480.405,A -85,B 0,C 180,E1 -2238.295,E2 -2238.295} C_VEL
LIN {X 0,Y 573.578,Z 492.648,A -85,B 0,C 180,E1 -2238.874,E2 -2238.874} C_VEL
LIN {X 0,Y 573.437,Z 504.218,A -85,B 0,C 180,E1 -2239.586,E2 -2239.586} C_VEL
LIN {X 0,Y 573.328,Z 514.615,A -85,B 0,C 180,E1 -2240.387,E2 -2240.387} C_VEL
LIN {X 0,Y 573.236,Z 523.081,A -85,B 0,C 180,E1 -2241.186,E2 -2241.186} C_VEL
LIN {X 0,Y 573.159,Z 530.97,A -85,B 0,C 180,E1 -2242.072,E2 -2242.072} C_VEL
LIN {X 0,Y 573.078,Z 538.899,A -85,B 0,C 180,E1 -2243.177,E2 -2243.177} C_VEL
LIN {X 0,Y 573.07,Z 545.686,A -85,B 0,C 180,E1 -2244.371,E2 -2244.371} C_VEL
LIN {X 0,Y 573.028,Z 550.377,A -85,B 0,C 180,E1 -2245.429,E2 -2245.429} C_VEL
LIN {X 0,Y 573.022,Z 553.961,A -85,B 0,C 180,E1 -2246.485,E2 -2246.485} C_VEL
